// TwinCAT 3 PLC project TcUnit
// Title: TcUnit
// Company: www.tcunit.org
// Author: Jakob Sagatowski and contributors
// ProjectVersion: 2026.7.18.1
// Description: TwinCAT unit testing framework. Documentation and examples are available at www.tcunit.org
// ProgramVersion: 3.1.4026.21
// libraries:
//   Base, * (Photara)
//   SysDir, * (System)
//   SysFile, * (System)
//   Tc2_Standard, * (Beckhoff Automation GmbH)
//   Tc2_System, * (Beckhoff Automation GmbH)
//   Tc2_Utilities, * (Beckhoff Automation GmbH)
//   Tc3_Module, * (Beckhoff Automation GmbH)
//   Base Interfaces,newest,System
// project tree:
//   DUTs/ E_AssertionType.TcDUT, E_XmlError.TcDUT (not stored), ST_AdsLogStringMessage.TcDUT (not stored), ST_AssertResult.TcDUT (not stored), ST_AssertResultInstances.TcDUT (not stored), ST_AssertArrayResult.TcDUT (not stored), ST_AssertArrayResultInstances.TcDUT (not stored), ST_TestCaseResult.TcDUT (not stored), ST_TestSuiteResult.TcDUT, ST_TestSuiteResults.TcDUT, U_ExpectedOrActual.TcDUT (not stored), E_WaitType.TcDUT, ST_TimedTestState.TcDUT, ST_TimedTestResult.TcDUT
//   GVLs/ GVL_Param_TcUnit.TcGVL (not stored), GVL_TcUnit.TcGVL (not stored)
//   ITFs/ I_AssertMessageFormatter.TcIO (not stored), I_TestResultLogger.TcIO (not stored), I_TestResults.TcIO (not stored)
//   POUs/ FB_AdsAssertMessageFormatter.TcPOU, FB_AdsLogStringMessageFifoQueue.TcPOU (not stored), FB_AdsTestResultLogger.TcPOU, FB_FileControl.TcPOU (not stored), FB_StreamBuffer.TcPOU (not stored), FB_xUnitXmlPublisher.TcPOU, FB_TestResults.TcPOU, FB_AdjustAssertFailureMessageToMax253CharLength.TcPOU (not stored), FB_AssertResultStatic.TcPOU, FB_AssertArrayResultStatic.TcPOU, FB_TcUnitRunner.TcPOU, FB_Test.TcPOU (not stored), FB_TestSuite.TcPOU, FB_TimedTestSuite.TcPOU, FB_XmlControl.TcPOU (not stored)
//   POUs/Functions/ F_AnyToUnionValue.TcPOU (not stored), F_AnyTypeClassToString.TcPOU (not stored), F_AssertionTypeToString.TcPOU, F_GetCpuCounterAs64bit.TcPOU (not stored), F_GetTestSuiteNameFromTestInstancePath.TcPOU (not stored), F_IsAnyEqualToUnionValue.TcPOU (not stored), F_RemoveInstancePathAndProjectNameFromTestInstancePath.TcPOU (not stored), IS_TEST_FINISHED.TcPOU (not stored), RUN.TcPOU (not stored), RUN_IN_SEQUENCE.TcPOU (not stored), TCUNIT_ADSLOGSTR.TcPOU (not stored), TEST.TcPOU (not stored), TEST_FINISHED.TcPOU (not stored), TEST_FINISHED_NAMED.TcPOU (not stored), TEST_ORDERED.TcPOU (not stored)
//   POUs/Functions/WRITE_PROTECTED_/ WRITE_PROTECTED_BOOL.TcPOU (not stored), WRITE_PROTECTED_BYTE.TcPOU (not stored), WRITE_PROTECTED_DATE.TcPOU (not stored), WRITE_PROTECTED_DATE_AND_TIME.TcPOU (not stored), WRITE_PROTECTED_DINT.TcPOU (not stored), WRITE_PROTECTED_DWORD.TcPOU (not stored), WRITE_PROTECTED_INT.TcPOU (not stored), WRITE_PROTECTED_LREAL.TcPOU (not stored), WRITE_PROTECTED_REAL.TcPOU (not stored), WRITE_PROTECTED_SINT.TcPOU (not stored), WRITE_PROTECTED_STRING.TcPOU (not stored), WRITE_PROTECTED_WSTRING.TcPOU (not stored), WRITE_PROTECTED_TIME.TcPOU (not stored), WRITE_PROTECTED_TIME_OF_DAY.TcPOU (not stored), WRITE_PROTECTED_UDINT.TcPOU (not stored), WRITE_PROTECTED_UINT.TcPOU (not stored), WRITE_PROTECTED_ULINT.TcPOU (not stored), WRITE_PROTECTED_LWORD.TcPOU (not stored), WRITE_PROTECTED_LINT.TcPOU (not stored), WRITE_PROTECTED_USINT.TcPOU (not stored), WRITE_PROTECTED_WORD.TcPOU (not stored)
//   Version/ Global_Version.TcGVL

// ---- DUTs/E_AssertionType.TcDUT
{attribute 'qualified_only'}
{attribute 'strict'}
TYPE E_AssertionType :
(
    Type_UNDEFINED := 0,
    Type_ANY,

    // Primitive types
    Type_BOOL,
    Type_BYTE,
    Type_DATE,
    Type_DATE_AND_TIME,
    Type_DINT,
    Type_DWORD,
    Type_INT,
    Type_LINT,
    Type_LREAL,
    Type_LTIME,
    Type_LWORD,
    Type_REAL,
    Type_SINT,
    Type_STRING,
    Type_TIME,
    Type_TIME_OF_DAY,
    Type_UDINT,
    Type_UINT,
    Type_ULINT,
    Type_USINT,
    Type_WORD,
    Type_WSTRING,

    // Array types
    Type_Array2D_LREAL,
    Type_Array2D_REAL,
    Type_Array3D_LREAL,
    Type_Array3D_REAL,
    Type_Array_BOOL,
    Type_Array_BYTE,
    Type_Array_DINT,
    Type_Array_DWORD,
    Type_Array_INT,
    Type_Array_LINT,
    Type_Array_LREAL,
    Type_Array_LWORD,
    Type_Array_REAL,
    Type_Array_SINT,
    Type_Array_UDINT,
    Type_Array_UINT,
    Type_Array_ULINT,
    Type_Array_USINT,
    Type_Array_WORD,

    // Timed test types
    Type_TIMEOUT,
    Type_WAIT_MISUSE
) BYTE;
END_TYPE

// ---- DUTs/ST_TestSuiteResult.TcDUT
TYPE ST_TestSuiteResult :
STRUCT
    Name : T_MaxString; // Full class name
    Identity : UINT(0..GVL_Param_TcUnit.MaxNumberOfTestSuites); // Should be 0..GVL_Param_TcUnit.MaxNumberOfTestSuites-1 but gives unknown compiler error
    NumberOfTests : UINT(0..GVL_Param_TcUnit.MaxNumberOfTestsForEachTestSuite);
    NumberOfFailedTests : UINT(0..GVL_Param_TcUnit.MaxNumberOfTestsForEachTestSuite);
    NumberOfSkippedTests : UINT(0..GVL_Param_TcUnit.MaxNumberOfTestsForEachTestSuite);
    Duration : LREAL; // In seconds
    TestCaseResults : ARRAY[1..GVL_Param_TcUnit.MaxNumberOfTestsForEachTestSuite] OF ST_TestCaseResult;
END_STRUCT
END_TYPE

// ---- DUTs/ST_TestSuiteResults.TcDUT
TYPE ST_TestSuiteResults :
STRUCT
    // General test results
    NumberOfTestSuites : UINT; // The total number of test suites
    NumberOfTestCases : UDINT; // The total number of test cases (for all test suites)
    NumberOfSuccessfulTestCases : UDINT; // The total number of test cases that had all ASSERTS successful
    NumberOfFailedTestCases : UDINT; // The total number of test cases that had at least one ASSERT failed
    NumberOfSkippedTestCases : UDINT; // The total number of test cases that were skipped (disabled)
    Duration : LREAL; // Duration it took for all test suites to finish, in seconds

    // Test results for each individiual test suite
    TestSuiteResults : ARRAY[1..GVL_Param_TcUnit.MaxNumberOfTestSuites] OF ST_TestSuiteResult;
END_STRUCT
END_TYPE

// ---- DUTs/E_WaitType.TcDUT
{attribute 'qualified_only'}
{attribute 'strict'}
TYPE E_WaitType :
(
    None      := 0,
    // 'Duration', not 'Time': TIME is an IEC reserved word; the compiler accepts a
    // qualified_only member named Time, but the 4026 library packer NREs on any
    // E_WaitType.Time reference during Save-as-Library (found 2026-07-17)
    Duration  := 1,
    Condition := 2
);
END_TYPE

// ---- DUTs/ST_TimedTestState.TcDUT
TYPE ST_TimedTestState :
STRUCT
    tSafetyTimeout     : TIME;
    nSafetyStartTime   : LWORD;
    bSafetyTimedOut    : BOOL;
    bInitialized       : BOOL;

    nWaitStartTime     : LWORD;
    bWaitComplete      : BOOL;
    bConditionTimedOut : BOOL;
    eWaitType          : E_WaitType;
    tLatchedDuration   : TIME;
END_STRUCT
END_TYPE

// ---- DUTs/ST_TimedTestResult.TcDUT
TYPE ST_TimedTestResult :
STRUCT
    TestName           : T_MaxString;
    bIsFailed          : BOOL;
    bIsSkipped         : BOOL;
    bIsFinished        : BOOL;
    sFailureMessage    : T_MaxString;
    eFailureType       : E_AssertionType;
    nNumberOfAsserts   : UINT;
    lrDuration         : LREAL;
    stTimedState       : ST_TimedTestState;
END_STRUCT
END_TYPE

// ---- Version/Global_Version.TcGVL
{attribute 'TcGenerated'}
{attribute 'no-analysis'}
{attribute 'linkalways'}
// This function has been automatically generated from the project information.
VAR_GLOBAL CONSTANT
	{attribute 'const_non_replaced'}
	stLibVersion_TcUnit : ST_LibVersion := (iMajor := 2026, iMinor := 7, iBuild := 18, iRevision := 1, nFlags := 0, sVersion := '2026.7.18.1');
END_VAR

// ---- POUs/FB_AdsAssertMessageFormatter.TcPOU
(*
    This function block is responsible for printing the results of the assertions using the built-in
    ADSLOGSTR functionality provided by the Tc2_System library. This sends the result using ADS, which
    is consumed by the error list of Visual Studio.
*)
FUNCTION_BLOCK FB_AdsAssertMessageFormatter EXTENDS Base.FB_BaseStatic IMPLEMENTS I_AssertMessageFormatter

METHOD PUBLIC LogAssertFailure
VAR_INPUT
    Expected : T_MaxString;
    Actual : T_MaxString;
    Message : T_MaxString;
    TestInstancePath : T_MaxString;
END_VAR
VAR
    AdjustAssertFailureMessageToMax253CharLength : FB_AdjustAssertFailureMessageToMax253CharLength;
    TestInstancePathCleaned : T_MaxString;
    TestInstancePathFinal : T_MaxString;
    ReturnValue : DINT;
    TestInstancePathProcessed : T_MaxString;
    MessageProcessed : T_MaxString;
    TraceMessage : T_MaxString;
END_VAR
TestInstancePathCleaned := F_RemoveInstancePathAndProjectNameFromTestInstancePath(TestInstancePath);
TestInstancePathFinal := CONCAT(STR1 := 'FAILED TEST $'',
                                STR2 := TestInstancePathCleaned);
TestInstancePathFinal := CONCAT(STR1 := TestInstancePathFinal,
                                STR2 := '$'');

TestInstancePathFinal := CONCAT(STR1 := TestInstancePathFinal,
                                STR2 := ', EXP: ');
TestInstancePathFinal := CONCAT(STR1 := TestInstancePathFinal,
                                STR2 := Expected);
TestInstancePathFinal := CONCAT(STR1 := TestInstancePathFinal,
                                STR2 := ', ACT: ');
TestInstancePathFinal := CONCAT(STR1 := TestInstancePathFinal,
                                STR2 := Actual);
IF LEN(STR := Message) > 0 THEN
    TestInstancePathFinal := CONCAT(STR1 := TestInstancePathFinal,
                                    STR2 := ', MSG: %s');
END_IF

AdjustAssertFailureMessageToMax253CharLength(TestInstancePath := TestInstancePathFinal,
                                             TestMessage := Message,
                                             TestInstancePathProcessed => TestInstancePathProcessed,
                                             TestMessageProcessed => MessageProcessed);

GVL_TcUnit.AdsMessageQueue.WriteLog(MsgCtrlMask := ADSLOG_MSGTYPE_ERROR,
                                    MsgFmtStr := TestInstancePathProcessed,
                                    StrArg := MessageProcessed);

TraceMessage := CONCAT(STR1 := 'ASSERT FAIL $'', STR2 := TestInstancePathCleaned);
TraceMessage := CONCAT(STR1 := TraceMessage, STR2 := '$', EXP: ');
TraceMessage := CONCAT(STR1 := TraceMessage, STR2 := Expected);
TraceMessage := CONCAT(STR1 := TraceMessage, STR2 := ', ACT: ');
TraceMessage := CONCAT(STR1 := TraceMessage, STR2 := Actual);
IF LEN(STR := Message) > 0 THEN
    TraceMessage := CONCAT(STR1 := TraceMessage, STR2 := ', MSG: ');
    TraceMessage := CONCAT(STR1 := TraceMessage, STR2 := Message);
END_IF
TraceWithSeverity(Message := TraceMessage, Severity := Global.TcEventSeverity.Error);
END_METHOD

END_FUNCTION_BLOCK

// ---- POUs/FB_AdsTestResultLogger.TcPOU
(*
    This function block reports the results from the tests using the built-in ADSLOGSTR functionality
    provided by the Tc2_System library. This sends the result using ADS, which is consumed by the "Error List"
    of Visual Studio (which can print Errors, Warnings and Messages).
*)
FUNCTION_BLOCK FB_AdsTestResultLogger EXTENDS FB_BaseStatic IMPLEMENTS I_TestResultLogger
VAR
    TestResults : I_TestResults;

    PrintingTestSuiteResultNumber : UINT(1..GVL_Param_TcUnit.MaxNumberOfTestSuites);
    PrintingTestSuiteTrigger : R_TRIG;

    // This flag is set once the final end result has printed
    PrintedFinalTestResults : BOOL;

    // This flag is set once the test suites result have been printed
    PrintedTestSuitesResults : BOOL;
END_VAR

METHOD FB_init : BOOL
VAR_INPUT
	bInitRetains : BOOL; // if TRUE, the retain variables are initialized (warm start / cold start)
	bInCopyCode : BOOL;  // if TRUE, the instance afterwards gets moved into the copy code (online change)
    iTestResults : I_TestResults;
END_VAR
TestResults := iTestResults;
END_METHOD

METHOD PUBLIC LogTestSuiteResults
VAR
    TcUnitTestResults : REFERENCE TO ST_TestSuiteResults;
    StringToPrint : T_MaxString; 
    TestsInTestSuiteCounter : UINT(1..GVL_Param_TcUnit.MaxNumberOfTestsForEachTestSuite);
    MaxNumberOfTestsToPrint : UINT(1..GVL_Param_TcUnit.MaxNumberOfTestsForEachTestSuite);
END_VAR
VAR CONSTANT
    TEST_STATUS_SKIP : STRING := 'SKIP';
    TEST_STATUS_PASS : STRING := 'PASS';
    TEST_STATUS_FAIL : STRING := 'FAIL';
END_VAR
TcUnitTestResults REF= TestResults.GetTestSuiteResults();

IF PrintingTestSuiteResultNumber <= GVL_TcUnit.NumberOfInitializedTestSuites AND NOT PrintedTestSuitesResults THEN
    PrintingTestSuiteTrigger(CLK := GVL_TcUnit.TestSuiteAddresses[PrintingTestSuiteResultNumber]^.AreAllTestsFinished());
    IF PrintingTestSuiteTrigger.Q THEN
        StringToPrint := CONCAT(STR1 := '| Test suite ID=',
                                STR2 := UINT_TO_STRING(TcUnitTestResults.TestSuiteResults[PrintingTestSuiteResultNumber].Identity));
        StringToPrint := CONCAT(STR1 := StringToPrint,
                                STR2 :=  ' $'%s$'');

        // Print test suite name and ID
        GVL_TcUnit.AdsMessageQueue.WriteLog(MsgCtrlMask := ADSLOG_MSGTYPE_HINT,
                                            MsgFmtStr := StringToPrint,
                                            StrArg := TcUnitTestResults.TestSuiteResults[PrintingTestSuiteResultNumber].Name);

        // Print number of tests/number of failed tests in test suite
        StringToPrint := CONCAT(STR1 := '| ID=',
                                             STR2 := UINT_TO_STRING(TcUnitTestResults.TestSuiteResults[PrintingTestSuiteResultNumber].Identity));
        StringToPrint := CONCAT(STR1 := StringToPrint,
                                             STR2 := ' number of tests=');
        StringToPrint := CONCAT(STR1 := StringToPrint,
                                             STR2 := UINT_TO_STRING(TcUnitTestResults.TestSuiteResults[PrintingTestSuiteResultNumber].NumberOfTests));
        StringToPrint := CONCAT(STR1 := StringToPrint,
                                             STR2 := ', number of failed tests=');
        StringToPrint := CONCAT(STR1 := StringToPrint,
                                             STR2 := UINT_TO_STRING(TcUnitTestResults.TestSuiteResults[PrintingTestSuiteResultNumber].NumberOfFailedTests));
        StringToPrint := CONCAT(STR1 := StringToPrint,
                                             STR2 := ', duration=');
        StringToPrint := CONCAT(STR1 := StringToPrint,
                                             STR2 := LREAL_TO_STRING(TcUnitTestResults.TestSuiteResults[PrintingTestSuiteResultNumber].Duration));
											 
        GVL_TcUnit.AdsMessageQueue.WriteLog(MsgCtrlMask := ADSLOG_MSGTYPE_HINT,
                                            MsgFmtStr := StringToPrint,
                                            StrArg := '');

        // Print error if there are too many tests in the test suite
        IF (TcUnitTestResults.TestSuiteResults[PrintingTestSuiteResultNumber].NumberOfTests > GVL_Param_TcUnit.MaxNumberOfTestsForEachTestSuite) THEN
            MaxNumberOfTestsToPrint := GVL_Param_TcUnit.MaxNumberOfTestsForEachTestSuite;
        ELSE
            MaxNumberOfTestsToPrint := TcUnitTestResults.TestSuiteResults[PrintingTestSuiteResultNumber].NumberOfTests;
        END_IF

        // Iterate and print all tests in test suite
        FOR TestsInTestSuiteCounter := 1 TO MaxNumberOfTestsToPrint BY 1 DO
            // Print test name
            GVL_TcUnit.AdsMessageQueue.WriteLog(MsgCtrlMask := ADSLOG_MSGTYPE_HINT,
                                                MsgFmtStr := '| Test name=%s',
                                                StrArg := TcUnitTestResults.TestSuiteResults[PrintingTestSuiteResultNumber].TestCaseResults[TestsInTestSuiteCounter].TestName);
            // Print test class name
            GVL_TcUnit.AdsMessageQueue.WriteLog(MsgCtrlMask := ADSLOG_MSGTYPE_HINT,
                                                MsgFmtStr := '| Test class name=%s',
                                                StrArg := TcUnitTestResults.TestSuiteResults[PrintingTestSuiteResultNumber].TestCaseResults[TestsInTestSuiteCounter].TestClassName);

            // Print test result/status (SUCCESS, FAILED, SKIPPED) + number of assertions made
            IF TcUnitTestResults.TestSuiteResults[PrintingTestSuiteResultNumber].TestCaseResults[TestsInTestSuiteCounter].TestIsFailed THEN
                StringToPrint := CONCAT(STR1 := '| Test status=', STR2 := TEST_STATUS_FAIL);
            ELSIF TcUnitTestResults.TestSuiteResults[PrintingTestSuiteResultNumber].TestCaseResults[TestsInTestSuiteCounter].TestIsSkipped THEN
                StringToPrint := CONCAT(STR1 := '| Test status=', STR2 := TEST_STATUS_SKIP);
            ELSE
                StringToPrint := CONCAT(STR1 := '| Test status=', STR2 := TEST_STATUS_PASS);
            END_IF

            StringToPrint := CONCAT(STR1 := StringToPrint, STR2 := ', number of asserts=');
            StringToPrint := CONCAT(STR1 := StringToPrint, STR2 :=
                                                 UINT_TO_STRING(TcUnitTestResults.TestSuiteResults[PrintingTestSuiteResultNumber].TestCaseResults[TestsInTestSuiteCounter].NumberOfAsserts));
            StringToPrint := CONCAT(STR1 := StringToPrint, STR2 := ', duration=');
            StringToPrint := CONCAT(STR1 := StringToPrint, STR2 :=
                                                 LREAL_TO_STRING(TcUnitTestResults.TestSuiteResults[PrintingTestSuiteResultNumber].TestCaseResults[TestsInTestSuiteCounter].Duration));												 
            GVL_TcUnit.AdsMessageQueue.WriteLog(MsgCtrlMask := ADSLOG_MSGTYPE_HINT,
                                                MsgFmtStr := StringToPrint,
                                                StrArg := '');

            // Print assertion/failure message (if existing)
            IF (LEN(STR := TcUnitTestResults.TestSuiteResults[PrintingTestSuiteResultNumber].TestCaseResults[TestsInTestSuiteCounter].FailureMessage) > 0) THEN
                GVL_TcUnit.AdsMessageQueue.WriteLog(MsgCtrlMask := ADSLOG_MSGTYPE_HINT,
                                                    MsgFmtStr := '| Test assert message=%s',
                                                    StrArg := TcUnitTestResults.TestSuiteResults[PrintingTestSuiteResultNumber].TestCaseResults[TestsInTestSuiteCounter].FailureMessage);
            END_IF

            // Print assertion/failure type (if existing)
            IF TcUnitTestResults.TestSuiteResults[PrintingTestSuiteResultNumber].TestCaseResults[TestsInTestSuiteCounter].FailureType <> E_AssertionType.Type_UNDEFINED THEN
                GVL_TcUnit.AdsMessageQueue.WriteLog(MsgCtrlMask := ADSLOG_MSGTYPE_HINT,
                                                    MsgFmtStr := '| Test assert type=%s',
                                                    StrArg := F_AssertionTypeToString(AssertionType :=
                                                        TcUnitTestResults.TestSuiteResults[PrintingTestSuiteResultNumber].TestCaseResults[TestsInTestSuiteCounter].FailureType));
            END_IF
        END_FOR

        // Print error message if there are too many tests in the test suite
        IF (TcUnitTestResults.TestSuiteResults[PrintingTestSuiteResultNumber].NumberOfTests > GVL_Param_TcUnit.MaxNumberOfTestsForEachTestSuite) THEN
            GVL_TcUnit.AdsMessageQueue.WriteLog(MsgCtrlMask := ADSLOG_MSGTYPE_ERROR,
                                                MsgFmtStr := 'Tests failed because the number of tests (%s',
                                                StrArg := CONCAT(STR1 := TO_STRING(TcUnitTestResults.TestSuiteResults[PrintingTestSuiteResultNumber].NumberOfTests),
                                                                              STR2 := CONCAT(STR1 := ') in the test suite $'',
                                                                                                          STR2 := CONCAT(STR1 := TcUnitTestResults.TestSuiteResults[PrintingTestSuiteResultNumber].Name,
                                                                                                                                      STR2 := CONCAT(STR1 := '$' are more than is defined in parameter $'GVL_Param_TcUnit.MaxNumberOfTestsForEachTestSuite$' (',
                                                                                                                                                                  STR2 := CONCAT(STR1 := UINT_TO_STRING(GVL_Param_TcUnit.MaxNumberOfTestsForEachTestSuite),
                                                                                                                                                                                              STR2 := '). Please increase this parameter.'))))));
            TraceWithSeverity(
                Message := CONCAT('Test count overflow in suite: ',
                           CONCAT(TcUnitTestResults.TestSuiteResults[PrintingTestSuiteResultNumber].Name,
                           CONCAT(' (', CONCAT(UINT_TO_STRING(TcUnitTestResults.TestSuiteResults[PrintingTestSuiteResultNumber].NumberOfTests),
                           CONCAT(' > ', CONCAT(UINT_TO_STRING(GVL_Param_TcUnit.MaxNumberOfTestsForEachTestSuite), ')')))))),
                Severity := Global.TcEventSeverity.Error);
        END_IF

        IF PrintingTestSuiteResultNumber = GVL_TcUnit.NumberOfInitializedTestSuites THEN
            PrintedTestSuitesResults := TRUE;
        ELSE
            PrintingTestSuiteResultNumber := PrintingTestSuiteResultNumber + 1;
        END_IF
        PrintingTestSuiteTrigger(CLK := FALSE); // Reset trigger
    END_IF
END_IF

// Log end results once all test suites have finished running
IF (GVL_TcUnit.NumberOfInitializedTestSuites = 0 OR PrintingTestSuiteResultNumber = GVL_TcUnit.NumberOfInitializedTestSuites)
    AND NOT PrintedFinalTestResults AND TestResults.GetAreTestResultsAvailable() THEN
    GVL_TcUnit.AdsMessageQueue.WriteLog(MsgCtrlMask := ADSLOG_MSGTYPE_ERROR,
                                        MsgFmtStr := '%s',
                                        StrArg := '| ==========TESTS FINISHED RUNNING==========');
    GVL_TcUnit.AdsMessageQueue.WriteLog(MsgCtrlMask := ADSLOG_MSGTYPE_ERROR,
                                        MsgFmtStr := '| Test suites: %s',
                                        StrArg := UINT_TO_STRING(TcUnitTestResults.NumberOfTestSuites));
    GVL_TcUnit.AdsMessageQueue.WriteLog(MsgCtrlMask := ADSLOG_MSGTYPE_ERROR,
                                        MsgFmtStr := '| Tests: %s',
                                        StrArg := UDINT_TO_STRING(TcUnitTestResults.NumberOfTestCases));
    GVL_TcUnit.AdsMessageQueue.WriteLog(MsgCtrlMask := ADSLOG_MSGTYPE_ERROR,
                                        MsgFmtStr := '| Successful tests: %s',
                                        StrArg := UDINT_TO_STRING(TcUnitTestResults.NumberOfSuccessfulTestCases));
    GVL_TcUnit.AdsMessageQueue.WriteLog(MsgCtrlMask := ADSLOG_MSGTYPE_ERROR,
                                        MsgFmtStr := '| Failed tests: %s',
                                        StrArg := UDINT_TO_STRING(TcUnitTestResults.NumberOfFailedTestCases));
    GVL_TcUnit.AdsMessageQueue.WriteLog(MsgCtrlMask := ADSLOG_MSGTYPE_ERROR,
                                        MsgFmtStr := '| Skipped tests: %s',
                                        StrArg := UDINT_TO_STRING(TcUnitTestResults.NumberOfSkippedTestCases));
    GVL_TcUnit.AdsMessageQueue.WriteLog(MsgCtrlMask := ADSLOG_MSGTYPE_ERROR,
                                        MsgFmtStr := '| Duration: %s',
                                        StrArg := LREAL_TO_STRING(TcUnitTestResults.Duration));                                        
    GVL_TcUnit.AdsMessageQueue.WriteLog(MsgCtrlMask := ADSLOG_MSGTYPE_ERROR,
                                        MsgFmtStr := '%s',
                                        StrArg := '| ======================================');

    TraceWithSeverity(
        Message := CONCAT('TESTS FINISHED - ',
                   CONCAT(UINT_TO_STRING(TcUnitTestResults.NumberOfTestSuites),
                   CONCAT(' suites, ',
                   CONCAT(UDINT_TO_STRING(TcUnitTestResults.NumberOfTestCases),
                   CONCAT(' tests, ',
                   CONCAT(UDINT_TO_STRING(TcUnitTestResults.NumberOfSuccessfulTestCases),
                   CONCAT(' passed, ',
                   CONCAT(UDINT_TO_STRING(TcUnitTestResults.NumberOfFailedTestCases),
                   CONCAT(' failed, ',
                   CONCAT(UDINT_TO_STRING(TcUnitTestResults.NumberOfSkippedTestCases), ' skipped')))))))))),
        Severity := Global.TcEventSeverity.Info);

    // Flush JSON event log so ToolPackageManager can read results immediately
    Base.GVL_System.FileHandlerJson.RequestFlush();

    PrintedFinalTestResults := TRUE;
END_IF
END_METHOD

END_FUNCTION_BLOCK

// ---- POUs/Functions/F_AssertionTypeToString.TcPOU
(* Since TwinCAT 3.1.4024.x it's possible to do TO_STRING on enumerations,
   but for backward compability we need to do it manually *)
FUNCTION F_AssertionTypeToString : T_MaxString
VAR_INPUT
    AssertionType : E_AssertionType;
END_VAR

CASE AssertionType OF
    E_AssertionType.Type_UNDEFINED :
        F_AssertionTypeToString := 'UNDEFINED';

    E_AssertionType.Type_ANY :
        F_AssertionTypeToString := 'ANY';

    (* Primitive types *)
    E_AssertionType.Type_BOOL :
        F_AssertionTypeToString := 'BOOL';

    E_AssertionType.Type_BYTE :
        F_AssertionTypeToString := 'BYTE';

    E_AssertionType.Type_DATE :
        F_AssertionTypeToString := 'DATE';

    E_AssertionType.Type_DATE_AND_TIME :
        F_AssertionTypeToString := 'DATE_AND_TIME';

    E_AssertionType.Type_DINT :
        F_AssertionTypeToString := 'DINT';

    E_AssertionType.Type_DWORD :
        F_AssertionTypeToString := 'DWORD';

    E_AssertionType.Type_INT :
        F_AssertionTypeToString := 'INT';

    E_AssertionType.Type_LINT :
        F_AssertionTypeToString := 'LINT';

    E_AssertionType.Type_LREAL :
        F_AssertionTypeToString := 'LREAL';

    E_AssertionType.Type_LTIME :
        F_AssertionTypeToString := 'LTIME';

    E_AssertionType.Type_LWORD :
        F_AssertionTypeToString := 'LWORD';

    E_AssertionType.Type_REAL :
        F_AssertionTypeToString := 'REAL';

    E_AssertionType.Type_SINT :
        F_AssertionTypeToString := 'SINT';

    E_AssertionType.Type_STRING :
        F_AssertionTypeToString := 'STRING';

    E_AssertionType.Type_TIME :
        F_AssertionTypeToString := 'TIME';

    E_AssertionType.Type_TIME_OF_DAY :
        F_AssertionTypeToString := 'TIME_OF_DAY';

    E_AssertionType.Type_UDINT :
        F_AssertionTypeToString := 'UDINT';

    E_AssertionType.Type_UINT :
        F_AssertionTypeToString := 'UINT';

    E_AssertionType.Type_ULINT :
        F_AssertionTypeToString := 'ULINT';

    E_AssertionType.Type_USINT :
        F_AssertionTypeToString := 'USINT';

    E_AssertionType.Type_WORD :
        F_AssertionTypeToString := 'WORD';

    E_AssertionType.Type_WSTRING :
        F_AssertionTypeToString := 'WSTRING';


    (* Array types *)
    E_AssertionType.Type_Array2D_LREAL :
        F_AssertionTypeToString := 'Array2D_LREAL';

    E_AssertionType.Type_Array2D_REAL :
        F_AssertionTypeToString := 'Array2D_REAL';

    E_AssertionType.Type_Array3D_LREAL :
        F_AssertionTypeToString := 'Array3D_LREAL';

    E_AssertionType.Type_Array3D_REAL :
        F_AssertionTypeToString := 'Array3D_REAL';

    E_AssertionType.Type_Array_BOOL :
        F_AssertionTypeToString := 'Array_BOOL';

    E_AssertionType.Type_Array_BYTE :
        F_AssertionTypeToString := 'Array_BYTE';

    E_AssertionType.Type_Array_DINT :
        F_AssertionTypeToString := 'Array_DINT';

    E_AssertionType.Type_Array_DWORD :
        F_AssertionTypeToString := 'Array_DWORD';

    E_AssertionType.Type_Array_INT :
        F_AssertionTypeToString := 'Array_INT';

    E_AssertionType.Type_Array_LINT :
        F_AssertionTypeToString := 'Array_LINT';

    E_AssertionType.Type_Array_LREAL :
        F_AssertionTypeToString := 'Array_LREAL';

    E_AssertionType.Type_Array_LWORD :
        F_AssertionTypeToString := 'Array_LWORD';

    E_AssertionType.Type_Array_REAL :
        F_AssertionTypeToString := 'Array_REAL';

    E_AssertionType.Type_Array_SINT :
        F_AssertionTypeToString := 'Array_SINT';

    E_AssertionType.Type_Array_UDINT :
        F_AssertionTypeToString := 'Array_UDINT';

    E_AssertionType.Type_Array_UINT :
        F_AssertionTypeToString := 'Array_UINT';

    E_AssertionType.Type_Array_ULINT :
        F_AssertionTypeToString := 'Array_ULINT';

    E_AssertionType.Type_Array_USINT :
        F_AssertionTypeToString := 'Array_USINT';

    E_AssertionType.Type_Array_WORD :
        F_AssertionTypeToString := 'Array_WORD';

    (* Timed test types *)
    E_AssertionType.Type_TIMEOUT :
        F_AssertionTypeToString := 'TIMEOUT';

    E_AssertionType.Type_WAIT_MISUSE :
        F_AssertionTypeToString := 'WAIT_MISUSE';

    ELSE
        F_AssertionTypeToString := 'UNDEFINED';

END_CASE

END_FUNCTION

// ---- POUs/FB_xUnitXmlPublisher.TcPOU
// Publishes test results into an xUnit compatible Xml file
FUNCTION_BLOCK FB_xUnitXmlPublisher EXTENDS FB_BaseStatic IMPLEMENTS I_TestResultLogger
VAR
    // Dependency injection via FB_Init
    TestResults : I_TestResults;

    // File access mode
    AccessMode : SysFile.ACCESS_MODE := SysFile.AM_WRITE_PLUS;

    File : FB_FileControl;
    Xml : FB_XMLControl;
    BufferInitialised : BOOL := FALSE;
    Buffer : ARRAY [0..(GVL_Param_TcUnit.XUnitBufferSize - 1)] OF BYTE;
    WritingTestSuiteResultNumber : UINT(1..GVL_Param_TcUnit.MaxNumberOfTestSuites);
    PublishTrigger : R_TRIG;
END_VAR

(*
    Deletes the former file (if it exists).
    Opens the file, writes the buffer and closes it.
*)
METHOD PRIVATE DeleteOpenWriteClose : SysFile.SysTypes.RTS_IEC_RESULT;
VAR
    WriteResult : SysFile.SysTypes.RTS_IEC_RESULT;
END_VAR
DeleteOpenWriteClose := SysDir.CmpErrors.Errors.ERR_OK;
IF Initialised() THEN
    // Delete may fail if file doesn't exist yet (first run) — not a real error
    DeleteOpenWriteClose := MAX(DeleteOpenWriteClose, File.Delete(Filename := GVL_Param_TcUnit.xUnitFilePath));
    // Track Open/Write/Close separately for trace — these are the real errors
    WriteResult := File.Open(Filename := GVL_Param_TcUnit.xUnitFilePath, FileAccessMode := AccessMode);
    WriteResult := MAX(WriteResult, File.Write(BufferPointer := ADR(Buffer), Xml.Length));
    WriteResult := MAX(WriteResult, File.Close());
    DeleteOpenWriteClose := MAX(DeleteOpenWriteClose, WriteResult);
ELSE
    WriteResult := SysDir.CmpErrors.Errors.ERR_NOBUFFER;
    DeleteOpenWriteClose := WriteResult;
END_IF;

IF WriteResult <> SysDir.CmpErrors.Errors.ERR_OK THEN
    TraceWithSeverity(
        Message := CONCAT('xUnit file I/O failure: ', GVL_Param_TcUnit.xUnitFilePath),
        Severity := Global.TcEventSeverity.Error);
END_IF;
END_METHOD

(*
    FB_Init is always available implicitly AND it is used primarily FOR initialization.
    The return value is not evaluated. For a specific influence, you can also declare the
    methods explicitly and provide additional code there with the standard initialization
    code. You can evaluate the return value.
*)
METHOD FB_Init: BOOL
VAR_INPUT
    bInitRetains: BOOL; // TRUE: the retain variables are initialized (reset warm / reset cold)
    bInCopyCode: BOOL;  // TRUE: the instance will be copied to the copy code afterward (online change)
    iTestResults : I_TestResults; // Interface dependency injection
END_VAR
// Set buffer and flag
Xml.SetBuffer(PointerToBuffer := ADR(Buffer), SizeOfBuffer := SIZEOF(Buffer));

// Set buffer initialised
BufferInitialised := TRUE;

// Set testresult interface
THIS^.TestResults := iTestResults;
END_METHOD

METHOD PRIVATE Initialised : BOOL
Initialised := THIS^.BufferInitialised;
END_METHOD

(*
    This method is responsible for the entire generation of the output file. 
    The output of the xml writer is NOT beautified.

    When new data is available, feel free to add it to the report
*)
METHOD PUBLIC LogTestSuiteResults
VAR
    UnitTestResults : REFERENCE TO ST_TestSuiteResults;
    CurrentSuiteNumber : UINT;
    CurrentTestCount : UINT;
END_VAR
VAR CONSTANT
    TEST_STATUS_SKIP : STRING := 'SKIP';
    TEST_STATUS_PASS : STRING := 'PASS';
    TEST_STATUS_FAIL : STRING := 'FAIL';
END_VAR
UnitTestResults REF= TestResults.GetTestSuiteResults();

// Only publish once if "GVL_Param_TcUnit.xUnitEnablePublish" is enabled and all test results are stored.
PublishTrigger(CLK := (TestResults.GetAreTestResultsAvailable() AND GVL_Param_TcUnit.xUnitEnablePublish));
IF PublishTrigger.Q THEN

    // <?xml version="1.0" encoding="UTF-8"?>
    Xml.WriteDocumentHeader(Header := '<?xml version="1.0" encoding="UTF-8"?>');

    // <testsuites>  ('disabled' removed 2026-07-18: an empty string breaks JUnit
    //  parsers expecting an integer; skipped counts carry the information)
    Xml.NewTag('testsuites');
    Xml.NewParameter('failures', UDINT_TO_STRING(UnitTestResults.NumberOfFailedTestCases));
    (* 'tests' is the TOTAL testcase count; the previous successful-only value was a bug *)
    Xml.NewParameter('tests', UDINT_TO_STRING(UnitTestResults.NumberOfTestCases));
    Xml.NewParameter('skipped', UDINT_TO_STRING(UnitTestResults.NumberOfSkippedTestCases));
    Xml.NewParameter('time', LREAL_TO_STRING(UnitTestResults.Duration));

    FOR CurrentSuiteNumber := 1 TO UnitTestResults.NumberOfTestSuites BY 1 DO
        // <testsuite>
        Xml.NewTag('testsuite');
        Xml.NewParameter('id', UINT_TO_STRING(UnitTestResults.TestSuiteResults[CurrentSuiteNumber].Identity));
        Xml.NewParameter('name', UnitTestResults.TestSuiteResults[CurrentSuiteNumber].name);
        Xml.NewParameter('tests', UINT_TO_STRING(UnitTestResults.TestSuiteResults[CurrentSuiteNumber].NumberOfTests));
        Xml.NewParameter('failures', UINT_TO_STRING(UnitTestResults.TestSuiteResults[CurrentSuiteNumber].NumberOfFailedTests));
        Xml.NewParameter('skipped', UINT_TO_STRING(UnitTestResults.TestSuiteResults[CurrentSuiteNumber].NumberOfSkippedTests));
        Xml.NewParameter('time', LREAL_TO_STRING(UnitTestResults.TestSuiteResults[CurrentSuiteNumber].Duration));

        FOR CurrentTestCount := 1 TO UnitTestResults.TestSuiteResults[CurrentSuiteNumber].NumberOfTests BY 1 DO
            // <testcase>
            Xml.NewTag('testcase');
            Xml.NewParameter('name', UnitTestResults.TestSuiteResults[CurrentSuiteNumber].TestCaseResults[CurrentTestCount].TestName);
            Xml.NewParameter('classname', UnitTestResults.TestSuiteResults[CurrentSuiteNumber].TestCaseResults[CurrentTestCount].TestClassName);
            Xml.NewParameter('time', LREAL_TO_STRING(UnitTestResults.TestSuiteResults[CurrentSuiteNumber].TestCaseResults[CurrentTestCount].Duration));

            IF UnitTestResults.TestSuiteResults[CurrentSuiteNumber].TestCaseResults[CurrentTestCount].TestIsFailed THEN
                Xml.NewParameter('status', TEST_STATUS_FAIL);
            ELSIF UnitTestResults.TestSuiteResults[CurrentSuiteNumber].TestCaseResults[CurrentTestCount].TestIsSkipped THEN
                Xml.NewParameter('status', TEST_STATUS_SKIP);
            ELSE
                Xml.NewParameter('status', TEST_STATUS_PASS);
            END_IF

            // Determine testcase fail, skip, or success
            IF UnitTestResults.TestSuiteResults[CurrentSuiteNumber].TestCaseResults[CurrentTestCount].FailureType <> E_AssertionType.Type_UNDEFINED THEN
                (* In case of fail
                    <failure message="Values differ" type="BYTE" />
                *)
                Xml.NewTag('failure');
                Xml.NewParameter('message', UnitTestResults.TestSuiteResults[CurrentSuiteNumber].TestCaseResults[CurrentTestCount].FailureMessage);
                Xml.NewParameter('type', F_AssertionTypeToString(UnitTestResults.TestSuiteResults[CurrentSuiteNumber].TestCaseResults[CurrentTestCount].FailureType));
                // Close failure tag
                Xml.CloseTag();
            ELSIF UnitTestResults.TestSuiteResults[CurrentSuiteNumber].TestCaseResults[CurrentTestCount].TestIsSkipped THEN
                (* JUnit consumers recognize a skipped testcase through a <skipped/>
                   child element, not a custom status attribute (kept for
                   backward compatibility) *)
                Xml.NewTag('skipped');
                Xml.CloseTag();
            ELSE
            // In case of success
            Xml.NewTagData('');

            END_IF
            // Close testcase tag
            Xml.CloseTag();

        END_FOR
        // Close testsuite tag
        Xml.CloseTag();

    END_FOR
    // Close testsuites
    Xml.CloseTag();

    // Delete, open, save and close the file
    DeleteOpenWriteClose();

    // Clear the internal buffer
    Xml.ClearBuffer();

    // Inform user
    GVL_TcUnit.AdsMessageQueue.WriteLog(MsgCtrlMask := ADSLOG_MSGTYPE_HINT,
                                        msgFmtStr := '%s',
                                        strArg := '| ==========TEST RESULTS EXPORTED===========');

    GVL_TcUnit.AdsMessageQueue.WriteLog(MsgCtrlMask := ADSLOG_MSGTYPE_HINT,
                                        msgFmtStr :=  '| Location: %s ',
                                        strArg := GVL_Param_TcUnit.xUnitFilePath);

    GVL_TcUnit.AdsMessageQueue.WriteLog(MsgCtrlMask := ADSLOG_MSGTYPE_HINT,
                                        MsgFmtStr := '%s',
                                        StrArg := '| ======================================');

    TraceWithSeverity(
        Message := CONCAT('xUnit XML exported to ', GVL_Param_TcUnit.xUnitFilePath),
        Severity := Global.TcEventSeverity.Info);
END_IF
END_METHOD

END_FUNCTION_BLOCK

// ---- POUs/FB_TestResults.TcPOU
// This function block holds results of the complete test run, i.e. results for all test suites
FUNCTION_BLOCK FB_TestResults IMPLEMENTS I_TestResults
VAR
    // Test results
    TestSuiteResults : ST_TestSuiteResults;

    // Misc variables
    StoringTestSuiteResultNumber : UINT(1..GVL_Param_TcUnit.MaxNumberOfTestSuites);
    StoringTestSuiteTrigger : R_TRIG;
    StoredTestSuiteResults : BOOL;
    StoredGeneralTestResults : BOOL;
    NumberOfTestsToAnalyse : UINT(1..GVL_Param_TcUnit.MaxNumberOfTestsForEachTestSuite);
END_VAR
VAR_TEMP
    TestSuiteName : T_MaxString;
    TestName : T_MaxString;

    TestsInTestSuiteCounter : UINT(1..GVL_Param_TcUnit.MaxNumberOfTestsForEachTestSuite);

    TestToBeStored : FB_Test;
    GeneralTestResultsTestSuitesCounter : UINT(1..GVL_Param_TcUnit.MaxNumberOfTestSuites);
END_VAR

// The body of the function block stores the test results
IF StoringTestSuiteResultNumber <= GVL_TcUnit.NumberOfInitializedTestSuites AND NOT StoredTestSuiteResults THEN
	StoringTestSuiteTrigger(CLK := GVL_TcUnit.TestSuiteAddresses[StoringTestSuiteResultNumber]^.AreAllTestsFinished());

    IF StoringTestSuiteTrigger.Q THEN
        // Remove everything except the program name + "." + test suite name
        TestSuiteName := F_RemoveInstancePathAndProjectNameFromTestInstancePath(TestInstancePath := GVL_TcUnit.TestSuiteAddresses[StoringTestSuiteResultNumber]^.GetInstancePath());

        // Store test suite name and ID
        TestSuiteResults.TestSuiteResults[StoringTestSuiteResultNumber].Name := TestSuiteName;
        TestSuiteResults.TestSuiteResults[StoringTestSuiteResultNumber].Identity := StoringTestSuiteResultNumber - 1;

        // Store number of tests in test suite
        TestSuiteResults.TestSuiteResults[StoringTestSuiteResultNumber].NumberOfTests :=
            GVL_TcUnit.TestSuiteAddresses[StoringTestSuiteResultNumber]^.GetNumberOfTests();

        // Store number of failed tests in test suite
        TestSuiteResults.TestSuiteResults[StoringTestSuiteResultNumber].NumberOfFailedTests :=
            GVL_TcUnit.TestSuiteAddresses[StoringTestSuiteResultNumber]^.GetNumberOfFailedTests();

        // Store number of skipped tests in test suite
        TestSuiteResults.TestSuiteResults[StoringTestSuiteResultNumber].NumberOfSkippedTests :=
            GVL_TcUnit.TestSuiteAddresses[StoringTestSuiteResultNumber]^.GetNumberOfSkippedTests();

        // Store the duration
        TestSuiteResults.TestSuiteResults[StoringTestSuiteResultNumber].Duration :=
            GVL_TcUnit.TestSuiteAddresses[StoringTestSuiteResultNumber]^.GetDuration();

        // Limit the test analyse to the max array limit of 'Tests[]' in FB_TestSuite
        NumberOfTestsToAnalyse := GVL_TcUnit.TestSuiteAddresses[StoringTestSuiteResultNumber]^.GetNumberOfTestsToAnalyse();

        // Iterate and print all tests in test suite
        FOR TestsInTestSuiteCounter := 1 TO NumberOfTestsToAnalyse BY 1 DO
            TestToBeStored := GVL_TcUnit.TestSuiteAddresses[StoringTestSuiteResultNumber]^.GetTestByPosition(TestsInTestSuiteCounter);
            // Store test name
            TestSuiteResults.TestSuiteResults[StoringTestSuiteResultNumber].TestCaseResults[TestsInTestSuiteCounter].TestName := TestToBeStored.GetName();

            // Store test class name
            TestSuiteResults.TestSuiteResults[StoringTestSuiteResultNumber].TestCaseResults[TestsInTestSuiteCounter].TestClassName :=
                F_RemoveInstancePathAndProjectNameFromTestInstancePath(GVL_TcUnit.TestSuiteAddresses[StoringTestSuiteResultNumber]^.GetInstancePath());

            // Store whether the test has failed
            TestSuiteResults.TestSuiteResults[StoringTestSuiteResultNumber].TestCaseResults[TestsInTestSuiteCounter].TestIsFailed :=
                TestToBeStored.IsFailed();

            // Store whether the test was skipped
            TestSuiteResults.TestSuiteResults[StoringTestSuiteResultNumber].TestCaseResults[TestsInTestSuiteCounter].TestIsSkipped :=
                TestToBeStored.IsSkipped();

            // Store the (first failed) assertion message
            TestSuiteResults.TestSuiteResults[StoringTestSuiteResultNumber].TestCaseResults[TestsInTestSuiteCounter].FailureMessage :=
                TestToBeStored.GetAssertionMessage();

            // Store the (first failed) assertion type
            TestSuiteResults.TestSuiteResults[StoringTestSuiteResultNumber].TestCaseResults[TestsInTestSuiteCounter].FailureType :=
                TestToBeStored.GetAssertionType();

            // Store number of assertions made
            TestSuiteResults.TestSuiteResults[StoringTestSuiteResultNumber].TestCaseResults[TestsInTestSuiteCounter].NumberOfAsserts :=
                TestToBeStored.GetNumberOfAssertions();

            // Store the duration of the test
            TestSuiteResults.TestSuiteResults[StoringTestSuiteResultNumber].TestCaseResults[TestsInTestSuiteCounter].Duration :=
                TestToBeStored.GetDuration();
        END_FOR

        IF StoringTestSuiteResultNumber = GVL_TcUnit.NumberOfInitializedTestSuites THEN
            StoredTestSuiteResults := TRUE;
        ELSE
            StoringTestSuiteResultNumber := StoringTestSuiteResultNumber + 1;
        END_IF
        StoringTestSuiteTrigger(CLK := FALSE); // Reset trigger
    END_IF
END_IF

(* If all test suites have finished running, store the general test results.
   Take care OF the special CASE where no tests have NOT yet been defined *)
IF GVL_TcUnit.NumberOfInitializedTestSuites = 0 AND (NOT StoredGeneralTestResults) THEN
    StoredGeneralTestResults := TRUE;
    StoredTestSuiteResults := TRUE;
ELSIF StoringTestSuiteResultNumber = GVL_TcUnit.NumberOfInitializedTestSuites AND_THEN
    GVL_TcUnit.TestSuiteAddresses[StoringTestSuiteResultNumber]^.AreAllTestsFinished() AND StoredTestSuiteResults AND (NOT StoredGeneralTestResults) THEN
    TestSuiteResults.NumberOfTestSuites := GVL_TcUnit.NumberOfInitializedTestSuites;
	GVL_TcUnit.Duration := LWORD_TO_LREAL(F_GetCpuCounterAs64bit(GVL_TcUnit.GetCpuCounter) - GVL_TcUnit.StartedAt) * GVL_TcUnit.HundredNanosecondToSecond; // Seconds
    TestSuiteResults.Duration := GVL_TcUnit.Duration;
    FOR GeneralTestResultsTestSuitesCounter := 1 TO GVL_TcUnit.NumberOfInitializedTestSuites BY 1 DO
        TestSuiteResults.NumberOfTestCases := TestSuiteResults.NumberOfTestCases + TestSuiteResults.TestSuiteResults[GeneralTestResultsTestSuitesCounter].NumberOfTests;
        (* A skipped test is not a successful test: total = passed + failed + skipped *)
        TestSuiteResults.NumberOfSuccessfulTestCases := TestSuiteResults.NumberOfSuccessfulTestCases +
                                                        (TestSuiteResults.TestSuiteResults[GeneralTestResultsTestSuitesCounter].NumberOfTests -
                                                         TestSuiteResults.TestSuiteResults[GeneralTestResultsTestSuitesCounter].NumberOfFailedTests -
                                                         TestSuiteResults.TestSuiteResults[GeneralTestResultsTestSuitesCounter].NumberOfSkippedTests);
        TestSuiteResults.NumberOfFailedTestCases := TestSuiteResults.NumberOfFailedTestCases + TestSuiteResults.TestSuiteResults[GeneralTestResultsTestSuitesCounter].NumberOfFailedTests;
        TestSuiteResults.NumberOfSkippedTestCases := TestSuiteResults.NumberOfSkippedTestCases + TestSuiteResults.TestSuiteResults[GeneralTestResultsTestSuitesCounter].NumberOfSkippedTests;
    END_FOR
    StoredGeneralTestResults := TRUE;
END_IF

// Returns whether the storing of the test results is finished
METHOD PUBLIC GetAreTestResultsAvailable : BOOL
GetAreTestResultsAvailable := (StoredTestSuiteResults AND StoredGeneralTestResults);
END_METHOD

METHOD PUBLIC GetTestSuiteResults : REFERENCE TO ST_TestSuiteResults;
GetTestSuiteResults REF=TestSuiteResults;
END_METHOD

END_FUNCTION_BLOCK

// ---- POUs/FB_AssertResultStatic.TcPOU
(*
    This function block is responsible for keeping track of which asserts that have been made. The reason we need to
    keep track of these is because if the user does the same assert twice (because of running a test suite over several
    PLC-cycles) we want to know it so we don't print several times (if the assert fails).
    An instance of an assert is keyed/identified with the following parameters as key:
    - Value of expected
    - Value of actual
    - Message (string)
    - Test instance path (string)
*)
FUNCTION_BLOCK FB_AssertResultStatic EXTENDS FB_BaseStatic
VAR
    // The total number of instances of each of the "AssertResults"
    AssertResults : ARRAY[1..GVL_Param_TcUnit.MaxNumberOfAssertsForEachTestSuite] OF ST_AssertResult;

    // The total number of unique asserts
    TotalAsserts : UINT := 0;

    // Function block to get the current task cycle
    GetCurrentTaskIndex : GETCURTASKINDEX;

    // The total number of instances of each of the "AssertResults"
    AssertResultInstances : ARRAY[1..GVL_Param_TcUnit.MaxNumberOfAssertsForEachTestSuite] OF ST_AssertResultInstances;

    // The last PLC cycle count
    CycleCount : UDINT;

    // Only run first cycle
    FirstCycleExecuted : BOOL;
END_VAR

METHOD PRIVATE AddAssertResult
VAR_INPUT
    ExpectedSize : UDINT;
    ExpectedTypeClass : IBaseLibrary.TypeClass;
    ExpectedValue : POINTER TO BYTE;
    ActualSize : UDINT;
    ActualTypeClass : IBaseLibrary.TypeClass;
    ActualValue : POINTER TO BYTE;
    Message : T_MaxString;
    TestInstancePath : T_MaxString;
END_VAR
VAR_INST
	AssertResultOverflow : BOOL := FALSE;
END_VAR
VAR
    sErrorString : T_MaxString;
END_VAR
IF TotalAsserts < GVL_Param_TcUnit.MaxNumberOfAssertsForEachTestSuite THEN
    TotalAsserts := TotalAsserts + 1;
    AssertResults[TotalAsserts].Expected := F_AnyToUnionValue(AnySize := ExpectedSize, AnyTypeClass := ExpectedTypeClass, AnyValue := ExpectedValue);
    AssertResults[TotalAsserts].Actual := F_AnyToUnionValue(AnySize := ActualSize, AnyTypeClass := ActualTypeClass, AnyValue := ActualValue);
    AssertResults[TotalAsserts].Message := Message;
    AssertResults[TotalAsserts].TestInstancePath := TestInstancePath;
ELSE
    IF NOT AssertResultOverflow THEN
        sErrorString := CONCAT(STR1 := F_GetTestSuiteNameFromTestInstancePath(TestInstancePath := TestInstancePath),
                               STR2 := '. Max number of assertions exceeded. Check parameter MaxNumberOfAssertsForEachTestSuite.');
		GVL_TcUnit.AdsMessageQueue.WriteLog(msgCtrlMask := ADSLOG_MSGTYPE_ERROR,
											msgFmtStr := sErrorString,
											strArg := '');
		TraceWithSeverity(
			Message := sErrorString,
			Severity := Global.TcEventSeverity.Error);
		AssertResultOverflow := TRUE;
	END_IF
END_IF
END_METHOD

METHOD PRIVATE CopyDetectionCountAndResetDetectionCountInThisCycle
VAR
    IteratorCounter : UINT;
END_VAR
FOR IteratorCounter := 1 TO GVL_Param_TcUnit.MaxNumberOfAssertsForEachTestSuite BY 1 DO
    AssertResultInstances[IteratorCounter].DetectionCount := AssertResultInstances[IteratorCounter].DetectionCountThisCycle;
    AssertResultInstances[IteratorCounter].DetectionCountThisCycle := 0;
END_FOR
END_METHOD

METHOD PRIVATE CreateAssertResultInstance
VAR_INPUT
    ExpectedSize : UDINT;
    ExpectedTypeClass : IBaseLibrary.TypeClass;
    ExpectedValue : POINTER TO BYTE;
    ActualSize : UDINT;
    ActualTypeClass : IBaseLibrary.TypeClass;
    ActualValue : POINTER TO BYTE;
    Message : T_MaxString;
    TestInstancePath : T_MaxString;
END_VAR
VAR
    IteratorCounter : UINT;
END_VAR
FOR IteratorCounter := 1 TO GVL_Param_TcUnit.MaxNumberOfAssertsForEachTestSuite BY 1 DO
    IF AssertResultInstances[IteratorCounter].DetectionCount = 0 AND
        AssertResultInstances[IteratorCounter].DetectionCountThisCycle = 0 THEN // Find first free spot
        AssertResultInstances[IteratorCounter].AssertResult.Expected := F_AnyToUnionValue(AnySize := ExpectedSize, AnyTypeClass := ExpectedTypeClass, AnyValue := ExpectedValue);
        AssertResultInstances[IteratorCounter].AssertResult.Actual := F_AnyToUnionValue(AnySize := ActualSize, AnyTypeClass := ActualTypeClass, AnyValue := ActualValue);
        AssertResultInstances[IteratorCounter].AssertResult.Message := Message;
        AssertResultInstances[IteratorCounter].AssertResult.TestInstancePath := TestInstancePath;
        AssertResultInstances[IteratorCounter].DetectionCountThisCycle := 1;
        EXIT;
    END_IF
END_FOR
END_METHOD

METHOD PRIVATE GetDetectionCount : UINT
VAR_INPUT
    ExpectedSize : UDINT;
    ExpectedTypeClass : IBaseLibrary.TypeClass;
    ExpectedValue : POINTER TO BYTE;
    ActualSize : UDINT;
    ActualTypeClass : IBaseLibrary.TypeClass;
    ActualValue : POINTER TO BYTE;
    Message : T_MaxString;
    TestInstancePath : T_MaxString;
END_VAR
VAR
    IteratorCounter : UINT;
END_VAR
FOR IteratorCounter := 1 TO GVL_Param_TcUnit.MaxNumberOfAssertsForEachTestSuite BY 1 DO
    IF F_IsAnyEqualToUnionValue(ExpectedOrActual := AssertResultInstances[IteratorCounter].AssertResult.Expected,
                                ExpectedOrActualSize := ExpectedSize,
                                ExpectedOrActualTypeClass := ExpectedTypeClass,
                                ExpectedOrActualValue := ExpectedValue) AND
       F_IsAnyEqualToUnionValue(ExpectedOrActual := AssertResultInstances[IteratorCounter].AssertResult.Actual,
                                ExpectedOrActualSize := ActualSize,
                                ExpectedOrActualTypeClass := ActualTypeClass,
                                ExpectedOrActualValue := ActualValue) AND
        AssertResultInstances[IteratorCounter].AssertResult.Message = Message AND
        AssertResultInstances[IteratorCounter].AssertResult.TestInstancePath = TestInstancePath THEN
        GetDetectionCount := AssertResultInstances[IteratorCounter].DetectionCount;
    END_IF
END_FOR
END_METHOD

METHOD PRIVATE GetDetectionCountThisCycle : UINT
VAR_INPUT
    ExpectedSize : UDINT;
    ExpectedTypeClass : IBaseLibrary.TypeClass;
    ExpectedValue : POINTER TO BYTE;
    ActualSize : UDINT;
    ActualTypeClass : IBaseLibrary.TypeClass;
    ActualValue : POINTER TO BYTE;
    Message : T_MaxString;
    TestInstancePath : T_MaxString;
END_VAR
VAR
    IteratorCounter : UINT;
END_VAR
FOR IteratorCounter := 1 TO GVL_Param_TcUnit.MaxNumberOfAssertsForEachTestSuite BY 1 DO
    IF F_IsAnyEqualToUnionValue(ExpectedOrActual := AssertResultInstances[IteratorCounter].AssertResult.Expected,
                                ExpectedOrActualSize := ExpectedSize,
                                ExpectedOrActualTypeClass := ExpectedTypeClass,
                                ExpectedOrActualValue := ExpectedValue) AND
       F_IsAnyEqualToUnionValue(ExpectedOrActual := AssertResultInstances[IteratorCounter].AssertResult.Actual,
                                ExpectedOrActualSize := ActualSize,
                                ExpectedOrActualTypeClass := ActualTypeClass,
                                ExpectedOrActualValue := ActualValue) AND
        AssertResultInstances[IteratorCounter].AssertResult.Message = Message AND
        AssertResultInstances[IteratorCounter].AssertResult.TestInstancePath = TestInstancePath THEN
        GetDetectionCountThisCycle := AssertResultInstances[IteratorCounter].DetectionCountThisCycle;
    END_IF
END_FOR
END_METHOD

METHOD INTERNAL GetNumberOfAssertsForTest : UINT
VAR_INPUT
    CompleteTestInstancePath : T_MaxString;
END_VAR
VAR
    Counter : UINT;
    NumberOfAsserts : UINT := 0;
END_VAR
IF TotalAsserts > 0 THEN
    FOR Counter := 1 TO TotalAsserts BY 1 DO
        IF AssertResults[Counter].TestInstancePath = CompleteTestInstancePath THEN
            NumberOfAsserts := NumberOfAsserts + 1;
        END_IF
    END_FOR
END_IF

GetNumberOfAssertsForTest := NumberOfAsserts;
END_METHOD

(*
    This method is called in every assert and returns whether this particular assert has already been called.
    The reason one would like to know whether this assert has already been reported or not is to not report it several
    times to any logging service. Because a test-suite can consist of several tests, and certain tests can require the
    test to run over several cycles it means that certain asserts could be called several times and thus we need to
    keep track of which asserts we've already reported. The user of the framework should not need to care for any of
    this and he/she should be able to call the asserts in any way they find suitable.

    To know what assert this is we need to check for the total combination of:
    - Test message
    - Test instance path
    - Expected value
    - Actual value
    Theoretically we can have a situation where a test has three different asserts, each and one with the same test
    message/test instance path/actual value/expected value but called within the same or different cycles. In order for
    us to handle all situations we need a simple algorithm that works according to:
    - Keep track of how many instances the combination of test message/test instance path/expected value/actual value
      we have. So for example, if we have called Assert(Exp := 5, Act := 5, 'Hello there', 'PRG.InstanceTestSuite.Test')
      two times in one cycle, we have two instances of that combination. This is done according to:
    - Iterate all existing reports.
      - If we have a new PLC-cycle, set the current detection-count to zero.
      - If new report does not match in any of the above fields, create it (together with current PLC-cycle).
        Also store the information that we have one instance of this combination and +1 on the detection-count.
      - If new report matches in all of the above, +1 in the detection-count. If this detection-count is larger than
        the stored detection-count for this combination, create a new report and add +1 to the storage of
        the detection-count.
*)
METHOD INTERNAL ReportResult
VAR_INPUT
    ExpectedSize : UDINT;
    ExpectedTypeClass : IBaseLibrary.TypeClass;
    ExpectedValue : POINTER TO BYTE;
    ActualSize : UDINT;
    ActualTypeClass : IBaseLibrary.TypeClass;
    ActualValue : POINTER TO BYTE;
    Message : T_MaxString;
    TestInstancePath : T_MaxString;
END_VAR
VAR_OUTPUT
    AlreadyReported : BOOL := FALSE;
END_VAR
VAR
    LocationIndex : UINT;
    DataTypesNotEquals : BOOL;
    DataSizeNotEquals : BOOL;
    DataContentNotEquals : BOOL;
    CurrentCycleCount : UDINT;
    IteratorCounter : UINT;
    DetectionCountTemp : UINT := 0;
    FoundOne : BOOL;
    AdditionalIdenticalAssert : BOOL;
END_VAR
IF NOT FirstCycleExecuted THEN
    GetCurrentTaskIndex();
    FirstCycleExecuted := TRUE;
END_IF

CurrentCycleCount := TwinCAT_SystemInfoVarList._TaskInfo[GetCurrentTaskIndex.index].CycleCount;
(* Is current cycle the same as the last call to this method?
   If not, reset the detection count *)
IF CurrentCycleCount <> CycleCount THEN
    CopyDetectionCountAndResetDetectionCountInThisCycle();
END_IF

FOR IteratorCounter := 1 TO TotalAsserts BY 1 DO
      IF F_IsAnyEqualToUnionValue(ExpectedOrActual := AssertResultInstances[IteratorCounter].AssertResult.Expected,
                                  ExpectedOrActualSize := ExpectedSize,
                                  ExpectedOrActualTypeClass := ExpectedTypeClass,
                                  ExpectedOrActualValue := ExpectedValue) AND
         F_IsAnyEqualToUnionValue(ExpectedOrActual := AssertResultInstances[IteratorCounter].AssertResult.Actual,
                                  ExpectedOrActualSize := ActualSize,
                                  ExpectedOrActualTypeClass := ActualTypeClass,
                                  ExpectedOrActualValue := ActualValue) AND
        AssertResultInstances[IteratorCounter].AssertResult.Message = Message AND
        AssertResultInstances[IteratorCounter].AssertResult.TestInstancePath = TestInstancePath THEN
            AssertResultInstances[IteratorCounter].DetectionCountThisCycle :=
                AssertResultInstances[IteratorCounter].DetectionCountThisCycle + 1;
            FoundOne := TRUE;
        IF AssertResultInstances[IteratorCounter].DetectionCountThisCycle >
            AssertResultInstances[IteratorCounter].DetectionCount THEN // This assert is new
            AdditionalIdenticalAssert := TRUE;
        END_IF
        EXIT;
    END_IF
END_FOR

// If not found anything, create the first
IF NOT FoundOne THEN
    // No existing match found, create a new entry
    AddAssertResult(ExpectedSize := ExpectedSize,
                    ExpectedTypeClass := ExpectedTypeClass,
                    ExpectedValue := ExpectedValue,
                    ActualSize := ActualSize,
                    ActualTypeClass := ActualTypeClass,
                    ActualValue := ActualValue,
                    Message := Message, TestInstancePath := TestInstancePath);

    CreateAssertResultInstance(ExpectedSize := ExpectedSize,
                               ExpectedTypeClass := ExpectedTypeClass,
                               ExpectedValue := ExpectedValue,
                               ActualSize := ActualSize,
                               ActualTypeClass := ActualTypeClass,
                               ActualValue := ActualValue,
                               Message := Message, TestInstancePath := TestInstancePath);
// An additional instance of this assert needs to be created
ELSIF AdditionalIdenticalAssert THEN
    AddAssertResult(ExpectedSize := ExpectedSize,
                    ExpectedTypeClass := ExpectedTypeClass,
                    ExpectedValue := ExpectedValue,
                    ActualSize := ActualSize,
                    ActualTypeClass := ActualTypeClass,
                    ActualValue := ActualValue,
                    Message := Message, TestInstancePath := TestInstancePath);
// In all other cases, this assert has already been reported, we don't need to do anything
ELSE
    AlreadyReported := TRUE;
END_IF

// Update the cycle count
CycleCount := TwinCAT_SystemInfoVarList._TaskInfo[GetCurrentTaskIndex.index].CycleCount;
END_METHOD

END_FUNCTION_BLOCK

// ---- POUs/FB_AssertArrayResultStatic.TcPOU
(*
    This function block is responsible for keeping track of which array-asserts that have been made.
    The reason we need to keep track of these is because if the user does the same assert twice
    (because of running a test suite over several PLC-cycles) we want to know it so we don't print several times
    (if the assert fails). An instance of an array-assert is keyed/identified with the following parameters as key:
    - Array-size (in bytes) of the expecteds
    - Datatype of the expecteds
    - Array-size (in bytes) of the actuals
    - Datatype of the actuals
    - Message (string)
    - Test instance path (string)
*)
FUNCTION_BLOCK FB_AssertArrayResultStatic EXTENDS FB_BaseStatic
VAR
    // The total number of instances of each of the "AssertArrayResults"
    AssertArrayResults : ARRAY[1..GVL_Param_TcUnit.MaxNumberOfAssertsForEachTestSuite] OF ST_AssertArrayResult;

    // The total number of unique asserts
    TotalArrayAsserts : UINT := 0;

    // Function block to get the current task cycle
    GetCurrentTaskIndex : GETCURTASKINDEX;

    // The total number of instances of each of the "AssertArrayResults"
    AssertArrayResultInstances : ARRAY[1..GVL_Param_TcUnit.MaxNumberOfAssertsForEachTestSuite] OF ST_AssertArrayResultInstances;

    // The last PLC cycle count
    CycleCount : UDINT;

    // Only run first cycle
    FirstCycleExecuted : BOOL;
END_VAR

METHOD PRIVATE AddAssertArrayResult
VAR_INPUT
    ExpectedsSize : UDINT;
    ExpectedsTypeClass : IBaseLibrary.TypeClass;
    ActualsSize : UDINT;
    ActualsTypeClass : IBaseLibrary.TypeClass;
    Message : T_MaxString;
    TestInstancePath : T_MaxString;
END_VAR
VAR_INST
	AssertResultOverflow : BOOL := FALSE;
END_VAR
VAR
    sErrorString : T_MaxString;
END_VAR
IF TotalArrayAsserts < GVL_Param_TcUnit.MaxNumberOfAssertsForEachTestSuite THEN
	TotalArrayAsserts := TotalArrayAsserts + 1;
	AssertArrayResults[TotalArrayAsserts].ExpectedsSize := ExpectedsSize;
	AssertArrayResults[TotalArrayAsserts].ExpectedsTypeClass := ExpectedsTypeClass;
	AssertArrayResults[TotalArrayAsserts].ActualsSize := ActualsSize;
	AssertArrayResults[TotalArrayAsserts].ActualsTypeClass := ActualsTypeClass;
	AssertArrayResults[TotalArrayAsserts].Message := Message;
	AssertArrayResults[TotalArrayAsserts].TestInstancePath := TestInstancePath;
ELSE
	IF NOT AssertResultOverflow THEN
        sErrorString := CONCAT(STR1 := F_GetTestSuiteNameFromTestInstancePath(TestInstancePath := TestInstancePath),
                               STR2 := '. Max number of assertions exceeded. Check parameter MaxNumberOfAssertsForEachTestSuite.');
		GVL_TcUnit.AdsMessageQueue.WriteLog(MsgCtrlMask := ADSLOG_MSGTYPE_ERROR,
											MsgFmtStr := sErrorString,
											StrArg := '');
		TraceWithSeverity(
			Message := sErrorString,
			Severity := Global.TcEventSeverity.Error);
		AssertResultOverflow := TRUE;
	END_IF
END_IF
END_METHOD

METHOD PRIVATE CopyDetectionCountAndResetDetectionCountInThisCycle
VAR
    IteratorCounter : UINT;
END_VAR
FOR IteratorCounter := 1 TO GVL_Param_TcUnit.MaxNumberOfAssertsForEachTestSuite BY 1 DO
    AssertArrayResultInstances[IteratorCounter].DetectionCount := AssertArrayResultInstances[IteratorCounter].DetectionCountThisCycle;
    AssertArrayResultInstances[IteratorCounter].DetectionCountThisCycle := 0;
END_FOR
END_METHOD

METHOD PRIVATE CreateAssertResultInstance
VAR_INPUT
    ExpectedsSize : UDINT;
    ExpectedsTypeClass : IBaseLibrary.TypeClass;
    ActualsSize : UDINT;
    ActualsTypeClass : IBaseLibrary.TypeClass;
    Message : T_MaxString;
    TestInstancePath : T_MaxString;
END_VAR
VAR
    IteratorCounter : UINT;
END_VAR
FOR IteratorCounter := 1 TO GVL_Param_TcUnit.MaxNumberOfAssertsForEachTestSuite BY 1 DO
    IF AssertArrayResultInstances[IteratorCounter].DetectionCount = 0 AND
        AssertArrayResultInstances[IteratorCounter].DetectionCountThisCycle = 0 THEN // Find first free spot
        AssertArrayResultInstances[IteratorCounter].AssertArrayResult.ExpectedsSize := ExpectedsSize;
        AssertArrayResultInstances[IteratorCounter].AssertArrayResult.ExpectedsTypeClass := ExpectedsTypeClass;
        AssertArrayResultInstances[IteratorCounter].AssertArrayResult.ActualsSize := ActualsSize;
        AssertArrayResultInstances[IteratorCounter].AssertArrayResult.ActualsTypeClass := ActualsTypeClass;
        AssertArrayResultInstances[IteratorCounter].AssertArrayResult.Message := Message;
        AssertArrayResultInstances[IteratorCounter].AssertArrayResult.TestInstancePath := TestInstancePath;
        AssertArrayResultInstances[IteratorCounter].DetectionCountThisCycle := 1;
        EXIT;
    END_IF
END_FOR
END_METHOD

METHOD PRIVATE GetDetectionCount : UINT
VAR_INPUT
    ExpectedsSize : UDINT;
    ExpectedsTypeClass : IBaseLibrary.TypeClass;
    ActualsSize : UDINT;
    ActualsTypeClass : IBaseLibrary.TypeClass;
    Message : T_MaxString;
    TestInstancePath : T_MaxString;
END_VAR
VAR
    IteratorCounter : UINT;
END_VAR
FOR IteratorCounter := 1 TO GVL_Param_TcUnit.MaxNumberOfAssertsForEachTestSuite BY 1 DO
    IF AssertArrayResultInstances[IteratorCounter].AssertArrayResult.ExpectedsSize = ExpectedsSize AND
       AssertArrayResultInstances[IteratorCounter].AssertArrayResult.ExpectedsTypeClass = ExpectedsTypeClass AND
       AssertArrayResultInstances[IteratorCounter].AssertArrayResult.ActualsSize = ActualsSize AND
       AssertArrayResultInstances[IteratorCounter].AssertArrayResult.ActualsTypeClass = ActualsTypeClass AND
       AssertArrayResultInstances[IteratorCounter].AssertArrayResult.Message = Message AND
       AssertArrayResultInstances[IteratorCounter].AssertArrayResult.TestInstancePath = TestInstancePath THEN
        GetDetectionCount := AssertArrayResultInstances[IteratorCounter].DetectionCount;
    END_IF
END_FOR
END_METHOD

METHOD PRIVATE GetDetectionCountThisCycle : UINT
VAR_INPUT
    ExpectedsSize : UDINT;
    ExpectedsTypeClass : IBaseLibrary.TypeClass;
    ActualsSize : UDINT;
    ActualsTypeClass : IBaseLibrary.TypeClass;
    Message : T_MaxString;
    TestInstancePath : T_MaxString;
END_VAR
VAR
    IteratorCounter : UINT;
END_VAR
FOR IteratorCounter := 1 TO GVL_Param_TcUnit.MaxNumberOfAssertsForEachTestSuite BY 1 DO
    IF AssertArrayResultInstances[IteratorCounter].AssertArrayResult.ExpectedsSize = ExpectedsSize AND
       AssertArrayResultInstances[IteratorCounter].AssertArrayResult.ExpectedsTypeClass = ExpectedsTypeClass AND
       AssertArrayResultInstances[IteratorCounter].AssertArrayResult.ActualsSize = ActualsSize AND
       AssertArrayResultInstances[IteratorCounter].AssertArrayResult.ActualsTypeClass = ActualsTypeClass AND
       AssertArrayResultInstances[IteratorCounter].AssertArrayResult.Message = Message AND
       AssertArrayResultInstances[IteratorCounter].AssertArrayResult.TestInstancePath = TestInstancePath THEN

        GetDetectionCountThisCycle := AssertArrayResultInstances[IteratorCounter].DetectionCountThisCycle;
    END_IF
END_FOR
END_METHOD

METHOD INTERNAL GetNumberOfArrayAssertsForTest : UINT
VAR_INPUT
    CompleteTestInstancePath : T_MaxString;
END_VAR
VAR
    Counter : UINT;
    NumberOfArrayAsserts : UINT := 0;
END_VAR
IF TotalArrayAsserts > 0 THEN
    FOR Counter := 1 TO TotalArrayAsserts BY 1 DO
        IF AssertArrayResults[Counter].TestInstancePath = CompleteTestInstancePath THEN
            NumberOfArrayAsserts := NumberOfArrayAsserts + 1;
        END_IF
    END_FOR
END_IF

GetNumberOfArrayAssertsForTest := NumberOfArrayAsserts;
END_METHOD

(*
    This method is called in every assert and returns whether this particular assert has already been called.
    The reason one would like to know whether this assert has already been reported or not is to not report it several
    times to any logging service. Because a test-suite can consist of several tests, and certain tests can require the
    test to run over several cycles it means that certain asserts could be called several times and thus we need to
    keep track of which asserts we've already reported. The user of the framework should not need to care for any of
    this and he/she should be able to call the asserts in any way they find suitable.

    To know what assert this is we need to check for the total combination of:
    - Test message
    - Test instance path
    - Expecteds size (in bytes)
    - Actuals size (in bytes)
    - Expecteds datatype
    - Actuals datatype
    Theoretically we can have a situation where a test has three different asserts, each and one with the same test
    message/test instance path/actuals size&datatype/expecteds size&datatype but called within the same or different
    cycles. In order for us to handle all situations we need a simple algorithm that works according to:
    - Keep track of how many instances the combination of test message/test instance path/expecteds size&datatype/
      actuals size&datatype we have. So for example, if we have called
      Assert(Exp := [5,4,3], Act := [5,4,3], 'Hello there', 'PRG.InstanceTestSuite.Test')
      two times in one cycle, we have two instances of that combination. This is done according to:
    - Iterate all existing reports.
      - If we have a new PLC-cycle, set the current detection-count to zero.
      - If new report does not match in any of the above fields, create it (together with current PLC-cycle).
        Also store the information that we have one instance of this combination and +1 on the detection-count.
      - If new report matches in all of the above, +1 in the detection-count. If this detection-count is larger than
        the stored detection-count for this combination, create a new report and add +1 to the storage of
        the detection-count.
*)
METHOD INTERNAL ReportResult
VAR_INPUT
    ExpectedsSize : UDINT;
    ExpectedsTypeClass : IBaseLibrary.TypeClass;
    ActualsSize : UDINT;
    ActualsTypeClass : IBaseLibrary.TypeClass;
    Message : T_MaxString;
    TestInstancePath : T_MaxString;
END_VAR
VAR_OUTPUT
    AlreadyReported : BOOL := FALSE;
END_VAR
VAR
    LocationIndex : UINT;
    DataTypesNotEquals : BOOL;
    DataSizeNotEquals : BOOL;
    DataContentNotEquals : BOOL;
    CurrentCycleCount : UDINT;
    IteratorCounter : UINT;
    DetectionCountTemp : UINT := 0;
    FoundOne : BOOL;
    AdditionalIdenticalAssert : BOOL;
END_VAR
IF NOT FirstCycleExecuted THEN
    GetCurrentTaskIndex();
    FirstCycleExecuted := TRUE;
END_IF

CurrentCycleCount := TwinCAT_SystemInfoVarList._TaskInfo[GetCurrentTaskIndex.index].CycleCount;
(* Is current cycle the same as the last call to this method?
   If not, reset the detection count *)
IF CurrentCycleCount <> CycleCount THEN
    CopyDetectionCountAndResetDetectionCountInThisCycle();
END_IF

FOR IteratorCounter := 1 TO TotalArrayAsserts BY 1 DO
    IF AssertArrayResultInstances[IteratorCounter].AssertArrayResult.ExpectedsSize = ExpectedsSize AND
        AssertArrayResultInstances[IteratorCounter].AssertArrayResult.ExpectedsTypeClass = ExpectedsTypeClass AND
        AssertArrayResultInstances[IteratorCounter].AssertArrayResult.ActualsSize = ActualsSize AND
        AssertArrayResultInstances[IteratorCounter].AssertArrayResult.ActualsTypeClass = ActualsTypeClass AND
        AssertArrayResultInstances[IteratorCounter].AssertArrayResult.Message = Message AND
        AssertArrayResultInstances[IteratorCounter].AssertArrayResult.TestInstancePath = TestInstancePath THEN
        AssertArrayResultInstances[IteratorCounter].DetectionCountThisCycle :=
            AssertArrayResultInstances[IteratorCounter].DetectionCountThisCycle + 1;
            FoundOne := TRUE;
        IF AssertArrayResultInstances[IteratorCounter].DetectionCountThisCycle >
                AssertArrayResultInstances[IteratorCounter].DetectionCount THEN // This assert is new
                AdditionalIdenticalAssert := TRUE;
        END_IF
        EXIT;
    END_IF
END_FOR

// If not found anything, create the first
IF NOT FoundOne THEN
    // No existing match found, create a new entry
    AddAssertArrayResult(ExpectedsSize := ExpectedsSize,
                         ExpectedsTypeClass := ExpectedsTypeClass,
                         ActualsSize := ActualsSize,
                         ActualsTypeClass := ActualsTypeClass,
                         Message := Message,
                         TestInstancePath := TestInstancePath);
    CreateAssertResultInstance(ExpectedsSize := ExpectedsSize,
                               ExpectedsTypeClass := ExpectedsTypeClass,
                               ActualsSize := ActualsSize,
                               ActualsTypeClass := ActualsTypeClass,
                               Message := Message,
                               TestInstancePath := TestInstancePath);
// An additional instance of this assert needs to be created
ELSIF AdditionalIdenticalAssert THEN
    AddAssertArrayResult(ExpectedsSize := ExpectedsSize,
                         ExpectedsTypeClass := ExpectedsTypeClass,
                         ActualsSize := ActualsSize,
                         ActualsTypeClass := ActualsTypeClass,
                         Message := Message,
                         TestInstancePath := TestInstancePath);
// In all other cases, this assert has already been reported, we don't need to do anything
ELSE
    AlreadyReported := TRUE;
END_IF

// Update the cycle count
CycleCount := TwinCAT_SystemInfoVarList._TaskInfo[GetCurrentTaskIndex.index].CycleCount;
END_METHOD

END_FUNCTION_BLOCK

// ---- POUs/FB_TcUnitRunner.TcPOU
// This function block is responsible for holding track of the tests and executing them.
FUNCTION_BLOCK FB_TcUnitRunner EXTENDS FB_BaseStatic
VAR
    // Indication of whether all test suites have reported that they are finished
    AllTestSuitesFinished : BOOL := FALSE;
    AllTestSuitesFinishedTrigger : R_TRIG;

    //Test result information
    TestResults : FB_TestResults;

    (* Prints the results to ADS so that Visual Studio can display the results.
       This test result formatter can be replaced with something else than ADS *)
    AdsTestResultLogger : FB_AdsTestResultLogger(TestResults);
    TestResultLogger : I_TestResultLogger := AdsTestResultLogger;

    (* If this flag is set, it means that some external event triggered the
       request to abort running the test suites *)
    AbortRunningTestSuites : BOOL;

    // Publishes a xUnit compatible XML file
    xUnitXmlPublisher : FB_xUnitXmlPublisher(TestResults);
    XmlTestResultPublisher : I_TestResultLogger := xUnitXmlPublisher;
END_VAR

(* This function sets a flag which makes the runner stop running the tests
   in the test suites *)
METHOD INTERNAL AbortRunningTestSuiteTests
AbortRunningTestSuites := TRUE;
(* Request semantics only; the runner emits 'TEST RUN ABORTED' when it honors the flag *)
TraceWithSeverity(
    Message := 'TEST RUN ABORT REQUESTED',
    Severity := Global.TcEventSeverity.Warning);
END_METHOD

// This runs all the test suites in parallel
METHOD INTERNAL RunTestSuiteTests
VAR
    Counter : UINT := 0;
    BusyPrinting : BOOL;
    (* We need to hold a temporary state of the statistics 
       as we don't consider the tests to be completely finished until all test suites have executed completely.
       The reason we want to do it this way is because a test suite can run over several cycles. Only once all tests
       are finished (which might take many cycles), do we gather correct statistics *)
    NumberOfTestSuitesFinished : UINT := 0;
END_VAR
IF GVL_TcUnit.StartedAt = 0 THEN
    GVL_TcUnit.StartedAt := F_GetCpuCounterAs64bit(GVL_TcUnit.GetCpuCounter);
    TraceWithSeverity(
        Message := CONCAT('TEST RUN STARTED - ',
                   CONCAT(UINT_TO_STRING(GVL_TcUnit.NumberOfInitializedTestSuites), ' suite(s), parallel execution')),
        Severity := Global.TcEventSeverity.Info);
END_IF

// Run TcUnit test suites
IF NOT AllTestSuitesFinished THEN
    IF GVL_TcUnit.NumberOfInitializedTestSuites = 0 THEN
        AllTestSuitesFinished := TRUE;
    ELSIF GVL_TcUnit.NumberOfInitializedTestSuites > 0 THEN
        FOR Counter := 1 TO GVL_TcUnit.NumberOfInitializedTestSuites BY 1 DO
            IF GVL_TcUnit.TestSuiteAddresses[Counter]^.AreAllTestsFinished() THEN
                NumberOfTestSuitesFinished := NumberOfTestSuitesFinished + 1;
            ELSE
                GVL_TcUnit.CurrentTestSuiteBeingCalled := GVL_TcUnit.TestSuiteAddresses[Counter];
				GVL_TcUnit.CurrentTestSuiteBeingCalled^.SetStartedAtIfNotSet(Timestamp := F_GetCpuCounterAs64bit(GVL_TcUnit.GetCpuCounter));
                GVL_TcUnit.CurrentTestSuiteBeingCalled^();
				// This is not an efficient way to set the duration
				IF GVL_TcUnit.TestSuiteAddresses[Counter]^.AreAllTestsFinished() THEN
					GVL_TcUnit.CurrentTestSuiteBeingCalled^.CalculateDuration(FinishedAt := F_GetCpuCounterAs64bit(GVL_TcUnit.GetCpuCounter));
				END_IF
            END_IF
        END_FOR
        (* Check if some event triggered an abortion of running the tests, in that case abort it now.
           This can be accomplished by setting the result of the test suites run to finished. *)
        IF AbortRunningTestSuites THEN
            (* Observed-abort effect trace: fires when the runner honors the abort flag,
               including raw online writes that never call AbortRunningTestSuiteTests().
               Naturally one-shot - the completion latch closes this branch next scan. *)
            TraceWithSeverity(
                Message := 'TEST RUN ABORTED',
                Severity := Global.TcEventSeverity.Warning);
            NumberOfTestSuitesFinished := GVL_TcUnit.NumberOfInitializedTestSuites;
        END_IF

        IF NumberOfTestSuitesFinished = GVL_TcUnit.NumberOfInitializedTestSuites THEN
            AllTestSuitesFinished := TRUE;
        END_IF
    END_IF
END_IF

AllTestSuitesFinishedTrigger(CLK := AllTestSuitesFinished);
(* Aborted and completed are distinct terminal outcomes: an honored abort already
   emitted TEST RUN ABORTED, so the normal completion trace is suppressed *)
IF AllTestSuitesFinishedTrigger.Q AND NOT AbortRunningTestSuites THEN
    TraceWithSeverity(
        Message := CONCAT('TEST RUN COMPLETED - ',
                   CONCAT(UINT_TO_STRING(GVL_TcUnit.NumberOfInitializedTestSuites), ' suite(s) finished')),
        Severity := Global.TcEventSeverity.Info);
END_IF

// Store test suite results continuously
TestResults();

// Log test suite results continuously
TestResultLogger.LogTestSuiteResults();

// Publish the xUnit Xml file once if enabled
XmlTestResultPublisher.LogTestSuiteResults();

// Run the buffered ADS logger
GVL_TcUnit.AdsMessageQueue();
END_METHOD

// This runs all the test suites in sequence (one after the other)
METHOD INTERNAL RunTestSuiteTestsInSequence
VAR_INPUT
    TimeBetweenTestSuitesExecution : TIME; // Time delay between a test suite is finished and the next test suite starts
END_VAR
VAR
    BusyPrinting : BOOL;
    (* We need to hold a temporary state of the statistics
       as we don't consider the tests to be completely finished until all test suites have executed completely.
       The reason we want to do it this way is because a test suite can run over several cycles. Only once all tests
       are finished (which might take many cycles), do we gather correct statistics *)
    NumberOfTestSuitesFinished : UINT := 0;
END_VAR
VAR_INST
    (* This variable holds which current test suite is being called, as we are running
       each one in a sequence (one by one) *)
     CurrentlyRunningTestSuite : UINT := 1;
     TimerBetweenExecutionOfTestSuites : TOF;
END_VAR
IF GVL_TcUnit.StartedAt = 0 THEN
    GVL_TcUnit.StartedAt := F_GetCpuCounterAs64bit(GVL_TcUnit.GetCpuCounter);
    TraceWithSeverity(
        Message := CONCAT('TEST RUN STARTED - ',
                   CONCAT(UINT_TO_STRING(GVL_TcUnit.NumberOfInitializedTestSuites), ' suite(s), sequential execution')),
        Severity := Global.TcEventSeverity.Info);
END_IF

TimerBetweenExecutionOfTestSuites(PT := TimeBetweenTestSuitesExecution);
// Run TcUnit test suites
IF NOT AllTestSuitesFinished THEN
    IF GVL_TcUnit.NumberOfInitializedTestSuites = 0 THEN
        AllTestSuitesFinished := TRUE;
    ELSIF GVL_TcUnit.NumberOfInitializedTestSuites > 0 THEN
        IF TimerBetweenExecutionOfTestSuites.Q THEN
            TimerBetweenExecutionOfTestSuites.IN := FALSE;
        END_IF
        IF GVL_TcUnit.TestSuiteAddresses[CurrentlyRunningTestSuite]^.AreAllTestsFinished() THEN
            IF CurrentlyRunningTestSuite <> GVL_TcUnit.NumberOfInitializedTestSuites THEN
                (* Address the finished suite directly: CurrentTestSuiteBeingCalled is
                   null until a suite has executed, e.g. when the first suite is empty *)
                GVL_TcUnit.TestSuiteAddresses[CurrentlyRunningTestSuite]^.CalculateDuration(FinishedAt := F_GetCpuCounterAs64bit(GVL_TcUnit.GetCpuCounter));
                CurrentlyRunningTestSuite := CurrentlyRunningTestSuite + 1;
                TimerBetweenExecutionOfTestSuites.IN := TRUE;
            ELSE
                (* The cursor is on the final suite and it reports finished - the whole
                   sequence is done. NumberOfTestSuitesFinished is a method VAR (reset
                   every call), so incremental counting can never reach the total; the
                   completion latch below fires from this assignment. Breadcrumb #19. *)
                NumberOfTestSuitesFinished := GVL_TcUnit.NumberOfInitializedTestSuites;
            END_IF
        ELSIF NOT TimerBetweenExecutionOfTestSuites.Q THEN
            GVL_TcUnit.CurrentTestSuiteBeingCalled := GVL_TcUnit.TestSuiteAddresses[CurrentlyRunningTestSuite];
			GVL_TcUnit.CurrentTestSuiteBeingCalled^.SetStartedAtIfNotSet(Timestamp := F_GetCpuCounterAs64bit(GVL_TcUnit.GetCpuCounter));
            GVL_TcUnit.CurrentTestSuiteBeingCalled^();
			// This is not an efficient way to set the duration
			IF GVL_TcUnit.TestSuiteAddresses[CurrentlyRunningTestSuite]^.AreAllTestsFinished() THEN
				GVL_TcUnit.CurrentTestSuiteBeingCalled^.CalculateDuration(FinishedAt := F_GetCpuCounterAs64bit(GVL_TcUnit.GetCpuCounter));
			END_IF
        END_IF
        (* Check if some event triggered an abortion of running the tests, in that case abort it now.
           This can be accomplished by setting the result of the test suites run to finished. *)
        IF AbortRunningTestSuites THEN
            (* Observed-abort effect trace: fires when the runner honors the abort flag,
               including raw online writes that never call AbortRunningTestSuiteTests().
               Naturally one-shot - the completion latch closes this branch next scan. *)
            TraceWithSeverity(
                Message := 'TEST RUN ABORTED',
                Severity := Global.TcEventSeverity.Warning);
            NumberOfTestSuitesFinished := GVL_TcUnit.NumberOfInitializedTestSuites;
        END_IF
        IF NumberOfTestSuitesFinished = GVL_TcUnit.NumberOfInitializedTestSuites THEN
            AllTestSuitesFinished := TRUE;
        END_IF
    END_IF
END_IF

AllTestSuitesFinishedTrigger(CLK := AllTestSuitesFinished);
(* Aborted and completed are distinct terminal outcomes: an honored abort already
   emitted TEST RUN ABORTED, so the normal completion trace is suppressed *)
IF AllTestSuitesFinishedTrigger.Q AND NOT AbortRunningTestSuites THEN
    TraceWithSeverity(
        Message := CONCAT('TEST RUN COMPLETED - ',
                   CONCAT(UINT_TO_STRING(GVL_TcUnit.NumberOfInitializedTestSuites), ' suite(s) finished')),
        Severity := Global.TcEventSeverity.Info);
END_IF

// Store test suite results continuously
TestResults();

// Log test suite results continuously
TestResultLogger.LogTestSuiteResults();

// Publish the xUnit Xml file once if enabled
XmlTestResultPublisher.LogTestSuiteResults();

// Run the buffered ADS logger
GVL_TcUnit.AdsMessageQueue();
END_METHOD

END_FUNCTION_BLOCK

// ---- POUs/FB_TestSuite.TcPOU
(* This function block is responsible for holding the internal state of the test suite.
   Every test suite can have one or more tests, and every test can do one or more asserts.
   It's also responsible for providing all the assert-methods for asserting different data types.
   Only failed assertions are recorded.
*)
{attribute 'call_after_init'}
{attribute 'reflection'}
FUNCTION_BLOCK FB_TestSuite EXTENDS FB_BaseStatic
VAR
//     {attribute 'instance-path'}
//     {attribute 'noinit'}
//     InstancePath : T_MaxString;

    (* We need to have access to specific information of the current task that this test suite
       is executed in. This is for instance necessary when we need to know whether a test is
       defined already. The definition of a test that is defined already is that we call on it
       with the same name twice in the same cycle *)
    GetCurrentTaskIndex : GETCURTASKINDEX;

    NumberOfTests : UINT(0..GVL_Param_TcUnit.MaxNumberOfTestsForEachTestSuite) := 0;
    Tests : ARRAY[1..GVL_Param_TcUnit.MaxNumberOfTestsForEachTestSuite] OF FB_Test;
    (* Rising trigger of whether we have already notified the user of that the test name pointed to by the current
       position is a duplicate *)
    TestDuplicateNameTrigger : ARRAY[1..GVL_Param_TcUnit.MaxNumberOfTestsForEachTestSuite] OF R_TRIG;
    (* Last cycle count index for a specific test. Used to detect whether this test has already been defined in the
       current test suite *)
    TestCycleCountIndex : ARRAY[1..GVL_Param_TcUnit.MaxNumberOfTestsForEachTestSuite] OF UDINT;

    AssertResults : FB_AssertResultStatic;
    AssertArrayResults : FB_AssertArrayResultStatic;

    (* Prints the failed asserts to ADS so that Visual Studio can display the assert message.
       This assert formatter can be replaced with something else than ADS *)
    AdsAssertMessageFormatter : FB_AdsAssertMessageFormatter;
    AssertMessageFormatter : I_AssertMessageFormatter := AdsAssertMessageFormatter;

    (* Stores the CPU cycle count with 100ns precision. It also is an indication whether this 
       test suite has started running its tests (> 0 means it has started) *)
    StartedAt : LWORD;

    (* Duration it took to run all tests in this testsuite - including the overhead from TcUnit
       in seconds *)
    Duration : LREAL;

    // Number of ordered tests (created by TEST_ORDERED()) that this test suite contains
    NumberOfOrderedTests : UINT(0..GVL_Param_TcUnit.MaxNumberOfTestsForEachTestSuite);

    // One-shot flag to prevent repeated empty suite trace
    EmptySuiteTraced : BOOL;

END_VAR

METHOD INTERNAL AddTest : REFERENCE TO FB_Test
VAR_INPUT
    TestName : T_MaxString;
    IsTestOrdered : BOOL;
END_VAR
VAR
    IteratorCounter : UINT;
    ErrorMessage : T_MaxString;
    TestInstancePath : T_MaxString;
    FunctionCallResult : DINT;
    CycleCount : UDINT;
    TestWithThisNameAlreadyExists : BOOL := FALSE;
    LowerCasedTestName : T_MaxString;
    TrimmedTestName : T_MaxString;
    IgnoreCurrentTestCase : BOOL;
    NumberOfTestsToAnalyse : UINT(1..GVL_Param_TcUnit.MaxNumberOfTestsForEachTestSuite);
END_VAR
GVL_TcUnit.IgnoreCurrentTest := FALSE; // Reset the ignore current test flag

TrimmedTestName := F_LTrim(in := TestName);
TrimmedTestName := F_RTrim(in := TrimmedTestName);
LowerCasedTestName := F_ToLCase(in := TrimmedTestName);

// If test should be disabled, make sure to remove the "disabled_"-part of it from the test name
IF FIND(STR1 := LowerCasedTestName, STR2 := 'disabled_') = 1 THEN
    IgnoreCurrentTestCase := TRUE;
    TrimmedTestName := DELETE(STR := TrimmedTestName, LEN := LEN(STR := 'disabled_'), POS := 1);
END_IF

GetCurrentTaskIndex(); // Gets the task index of where this function block instance is being run in

(* Check if the test name already exists. Make sure there are no other tests with the same name already
   added for this test suite *)

CycleCount := TwinCAT_SystemInfoVarList._TaskInfo[GetCurrentTaskIndex.index].CycleCount;

// Limit the test analyse to the max array limit of 'Tests[]'
NumberOfTestsToAnalyse := GetNumberOfTestsToAnalyse();

// Iterate all the test names that up to this point have been added for this test suite
FOR IteratorCounter := 1 TO NumberOfTestsToAnalyse BY 1 DO
    IF Tests[IteratorCounter].GetName() = TrimmedTestName THEN
        TestWithThisNameAlreadyExists := TRUE;
        // Check if a test with this name has already been called in this PLC cycle
        IF TestCycleCountIndex[IteratorCounter] = CycleCount THEN
            GVL_TcUnit.IgnoreCurrentTest := TRUE;
            (* A test with this name already exists for this test suite and has already been called in this cycle.
               Send a message notification, but only if we have not done so already. *)
            TestDuplicateNameTrigger[IteratorCounter](CLK := TRUE);
            IF TestDuplicateNameTrigger[IteratorCounter].Q THEN // Rising edge detected. We have not reported this before
                TestInstancePath := F_RemoveInstancePathAndProjectNameFromTestInstancePath(TestInstancePath :=
                                                                                           GVL_TcUnit.CurrentTestSuiteBeingCalled^.GetInstancePath());
                ErrorMessage := 'Test with name $'%s$' already exists in test suite $'';
                ErrorMessage := CONCAT(STR1 := ErrorMessage, STR2 := TestInstancePath);
                ErrorMessage := CONCAT(STR1 := ErrorMessage, STR2 := '$'');
                GVL_TcUnit.AdsMessageQueue.WriteLog(MsgCtrlMask := ADSLOG_MSGTYPE_ERROR,
                                                    MsgFmtStr := ErrorMessage,
                                                    StrArg := TrimmedTestName);
                TraceWithSeverity(
                    Message := CONCAT('DUPLICATE TEST [', CONCAT(TrimmedTestName,
                               CONCAT('] in suite ', TestInstancePath))),
                    Severity := Global.TcEventSeverity.Warning);
            END_IF
        END_IF
        TestCycleCountIndex[IteratorCounter] := CycleCount;
    END_IF
END_FOR

IF NOT TestWithThisNameAlreadyExists THEN
    // Test has not been found. Add it.
    Tests[IteratorCounter].SetName(Name := TrimmedTestName);
    NumberOfTests := NumberOfTests + 1;
    TestCycleCountIndex[NumberOfTests] := CycleCount;
    IF IgnoreCurrentTestCase THEN
        Tests[IteratorCounter].SetSkipped();
        TraceWithSeverity(
            Message := CONCAT('TEST SKIPPED: ', TrimmedTestName),
            Severity := Global.TcEventSeverity.Info);
    END_IF

    // Extra information to be added if test is ordered (called by TEST_ORDERED())
    IF IsTestOrdered THEN
        NumberOfOrderedTests := NumberOfOrderedTests + 1;
        Tests[IteratorCounter].SetTestOrder(OrderNumber := NumberOfOrderedTests);
    END_IF
END_IF

// Check if this test should be disabled
IF IgnoreCurrentTestCase THEN
    GVL_TcUnit.IgnoreCurrentTest := TRUE;
    RETURN;
END_IF

AddTest REF= GetTestByName(TrimmedTestName);
END_METHOD

METHOD INTERNAL AddTestNameToInstancePath : T_MaxString
VAR_INPUT
    TestInstancePath : T_MaxString;
END_VAR
VAR
    CompleteTestInstancePath : T_MaxString;
END_VAR
CompleteTestInstancePath := CONCAT(STR1 := TestInstancePath, STR2 := '@');
AddTestNameToInstancePath := CONCAT(STR1 := CompleteTestInstancePath, STR2 := GVL_TcUnit.CurrentTestNameBeingCalled);
END_METHOD

METHOD PUBLIC AreAllTestsFinished : BOOL
VAR
    Counter : UINT;
    GetCurTaskIndex : GETCURTASKINDEX;
    NumberOfTestsToAnalyse : UINT(1..GVL_Param_TcUnit.MaxNumberOfTestsForEachTestSuite);
END_VAR
AreAllTestsFinished := FALSE;

IF NumberOfTests > 0 THEN
    AreAllTestsFinished := TRUE;
    // Limit the test analyse to the max array limit of 'Tests[]'
    NumberOfTestsToAnalyse := GetNumberOfTestsToAnalyse();
    // A test is considered finished if it is finished running (i.e. set by TEST_FINISHED) or if it is skipped/disabled
    FOR Counter := 1 TO NumberOfTestsToAnalyse BY 1 DO
        AreAllTestsFinished := AreAllTestsFinished AND (Tests[Counter].IsFinished() OR Tests[Counter].IsSkipped());
    END_FOR
END_IF

(* If we have been running at least one cycle and no tests are registered, it means that this testsuite is empty
   and doesn't contain any test cases. In that case, ignore this testsuite. *)
GetCurTaskIndex();
IF NumberOfTests = 0 AND NOT TwinCAT_SystemInfoVarList._TaskInfo[GetCurTaskIndex.index].FirstCycle AND StartedAt > 0 THEN
	AreAllTestsFinished := TRUE;
	IF NOT EmptySuiteTraced THEN
		TraceWithSeverity(
			Message := CONCAT('EMPTY TEST SUITE - ', InstancePath),
			Severity := Global.TcEventSeverity.Warning);
		EmptySuiteTraced := TRUE;
	END_IF
END_IF
END_METHOD

// Asserts that two LREAL 2D-arrays are equal to within a positive delta. If they are not, an assertion error is created.
METHOD PUBLIC AssertArray2dEquals_LREAL
VAR_IN_OUT
    Expecteds : ARRAY[*,*] OF LREAL; // LREAL 2d array with expected values
    Actuals : ARRAY[*,*] OF LREAL; // LREAL 2d array with actual values
END_VAR
VAR_INPUT
    Delta : LREAL; // The maximum delta between the value of expected and actual for which both numbers are still considered equal, proportional to the expected value in that array cell
    Message : T_MaxString; // The identifying message for the assertion error
END_VAR
VAR
    Equals : BOOL := TRUE;
    SizeEquals : BOOL := TRUE;
    ExpectedString : T_MaxString;
    ActualString : T_MaxString;
    AlreadyReported : BOOL;
    TestInstancePath : T_MaxString;
    DimensionIndex : USINT; // Index when looping through Dimensions
    LowerBoundExpecteds : ARRAY[1..2] OF DINT; // Lower bounds of Expecteds array in each dimension
    UpperBoundExpecteds : ARRAY[1..2] OF DINT; // Upper bounds of Expecteds array in each dimension
    LowerBoundActuals : ARRAY[1..2] OF DINT; // Lower bounds of Actuals array in each dimension
    UpperBoundActuals : ARRAY[1..2] OF DINT; // Upper bounds of Actuals array in each dimension
    SizeOfExpecteds : ARRAY[1..2] OF DINT; // Size of Expecteds array in each dimension
    SizeOfActuals : ARRAY[1..2] OF DINT; // Size of Actuals array in each dimension
    Offset : ARRAY[1..2] OF DINT; // Current Array index offsets from Lower Bound in each dimension
    ExpectedArrayIndex : ARRAY[1..2] OF DINT; // Array of current Expected array indexes when looping through arrays
    ActualArrayIndex : ARRAY[1..2] OF DINT; // Array of current Actual array indexes when looping through arrays
    Expected : LREAL; // Single expected value
    Actual : LREAL; // Single actual value
END_VAR
IF GVL_TcUnit.IgnoreCurrentTest OR GVL_TcUnit.CurrentTestIsFinished THEN
    RETURN;
END_IF

TestInstancePath := AddTestNameToInstancePath(FindTestSuiteInstancePath());

(* UPPER_BOUND and LOWER_BOUND require literals for their second parameter,
   so they can't be called in a dimension-based loop.
   Thus we copy the array dimensions into arrays which accept variable indexes *)
LowerBoundExpecteds[1] := LOWER_BOUND(Expecteds, 1);
UpperBoundExpecteds[1] := UPPER_BOUND(Expecteds, 1);
LowerBoundExpecteds[2] := LOWER_BOUND(Expecteds, 2);
UpperBoundExpecteds[2] := UPPER_BOUND(Expecteds, 2);
LowerBoundActuals[1] := LOWER_BOUND(Actuals, 1);
UpperBoundActuals[1] := UPPER_BOUND(Actuals, 1);
LowerBoundActuals[2] := LOWER_BOUND(Actuals, 2);
UpperBoundActuals[2] := UPPER_BOUND(Actuals, 2);

FOR DimensionIndex := 1 TO 2 DO
    SizeOfExpecteds[DimensionIndex] := ABS(UpperBoundExpecteds[DimensionIndex] - LowerBoundExpecteds[DimensionIndex]) + 1;
    SizeOfActuals[DimensionIndex] := ABS(UpperBoundActuals[DimensionIndex] - LowerBoundActuals[DimensionIndex]) + 1;

    IF SizeOfExpecteds[DimensionIndex] <> SizeOfActuals[DimensionIndex] THEN
        Equals := FALSE;
        SizeEquals := FALSE;
    END_IF
END_FOR

IF SizeEquals THEN
    (* Even though we know that both arrays are equal in size, the two arrays can start at two completely different
       indexes in each dimension, which needs to be taken into account. *)
    FOR Offset[1] := 0 TO SizeOfExpecteds[1] - 1 DO // Iterate Dimension 1
        FOR Offset[2] := 0 TO SizeOfExpecteds[2] - 1 DO // Iterate Dimension 2
            // Update index variables
            FOR DimensionIndex := 1 TO 2 DO
                ExpectedArrayIndex[DimensionIndex] := LowerBoundExpecteds[DimensionIndex] + Offset[DimensionIndex];
                ActualArrayIndex[DimensionIndex] := LowerBoundActuals[DimensionIndex] + Offset[DimensionIndex];
            END_FOR

            // Get array element values
            Expected := Expecteds[ExpectedArrayIndex[1], ExpectedArrayIndex[2]];
            Actual := Actuals[ActualArrayIndex[1], ActualArrayIndex[2]]; 

            IF ABS(Expected - Actual) > Delta THEN
                Equals := FALSE;
                EXIT;
            END_IF
        END_FOR

        // Check for loop bailout
        IF NOT Equals THEN
            EXIT;
        END_IF
    END_FOR
END_IF

AssertArrayResults.ReportResult(ExpectedsSize := DINT_TO_UDINT(SizeOfExpecteds[1] * SizeOfExpecteds[2]),
                                ExpectedsTypeClass := IBaseLibrary.TypeClass.TYPE_LREAL,
                                ActualsSize := DINT_TO_UDINT(SizeOfActuals[1] * SizeOfActuals[2]),
                                ActualsTypeClass := IBaseLibrary.TypeClass.TYPE_LREAL,
                                Message := Message,
                                TestInstancePath := TestInstancePath,
                                AlreadyReported => AlreadyReported);

IF NOT AlreadyReported AND NOT Equals THEN
    SetTestFailed(AssertionType := E_AssertionType.Type_Array2D_LREAL,
                  AssertionMessage := Message);

    IF NOT SizeEquals THEN
        Message := CONCAT(STR1 := Message, STR2 := ', size of arrays not matching.');
        ExpectedString := 'SIZE = [';
        ExpectedString := CONCAT(STR1 := ExpectedString,STR2 := DINT_TO_STRING(LowerBoundExpecteds[1]));
        ExpectedString := CONCAT(STR1 := ExpectedString, STR2 := '..');
        ExpectedString := CONCAT(STR1 := ExpectedString, STR2 := DINT_TO_STRING(UpperBoundExpecteds[1]));
        ExpectedString := CONCAT(STR1 := ExpectedString, STR2 := ',');
        ExpectedString := CONCAT(STR1 := ExpectedString, STR2 := DINT_TO_STRING(LowerBoundExpecteds[2]));
        ExpectedString := CONCAT(STR1 := ExpectedString, STR2 := '..');
        ExpectedString := CONCAT(STR1 := ExpectedString, STR2 := DINT_TO_STRING(UpperBoundExpecteds[2]));
        ExpectedString := CONCAT(STR1 := ExpectedString, STR2 := '] (');
        ExpectedString := CONCAT(STR1 := ExpectedString, STR2 := DINT_TO_STRING(SizeOfExpecteds[1]));
        ExpectedString := CONCAT(STR1 := ExpectedString, STR2 := 'x');
        ExpectedString := CONCAT(STR1 := ExpectedString, STR2 := DINT_TO_STRING(SizeOfExpecteds[2]));
        ExpectedString := CONCAT(STR1 := ExpectedString, STR2 := ')');

